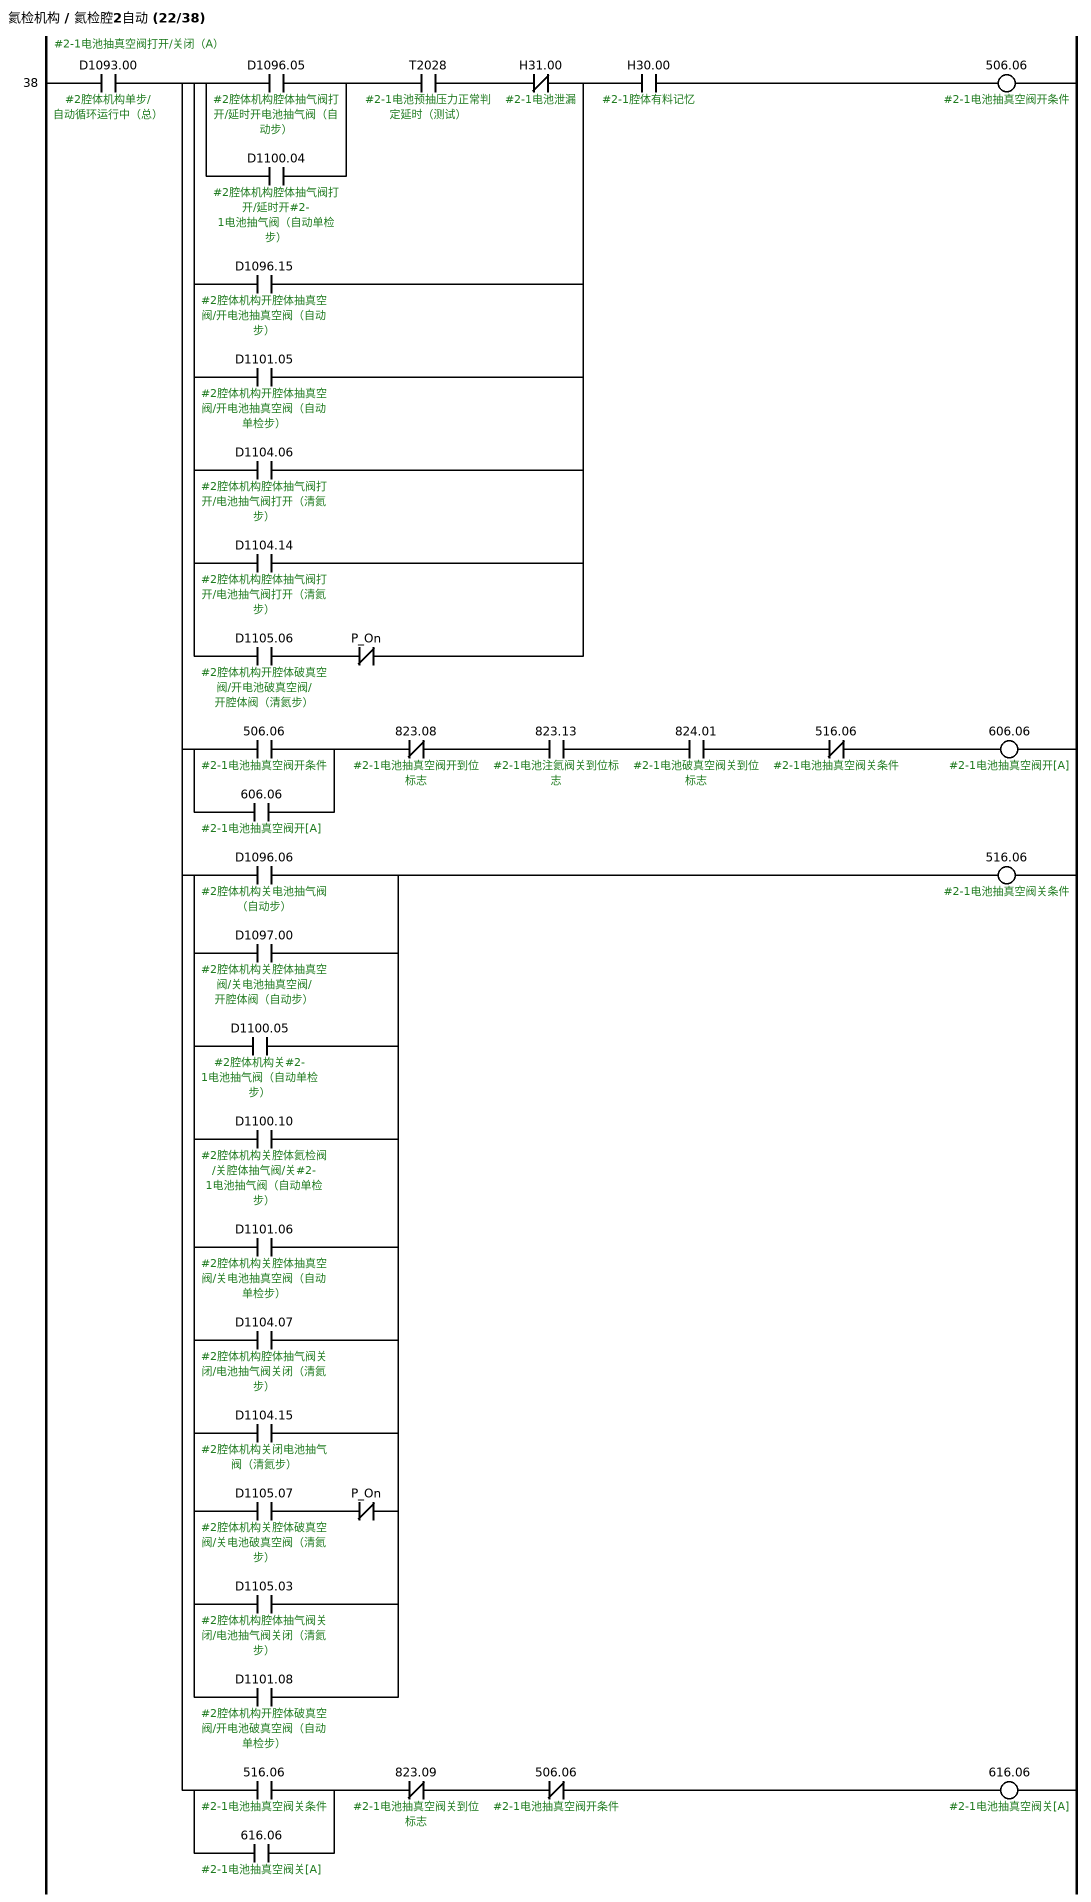
; [picture p264: 氦检机构 / 氦检腔2自动, rungs 38-38]
; rung 38: #2-1电池抽真空阀打开/关闭（A）
LD D1093.00  ; #2腔体机构单步/自动循环运行中（总）
OUT TR0
LD D1096.05  ; #2腔体机构腔体抽气阀打开/延时开电池抽气阀（自动步）
OR D1100.04  ; #2腔体机构腔体抽气阀打开/延时开#2-1电池抽气阀（自动单检步）
AND T2028  ; #2-1电池预抽压力正常判定延时（测试）
ANDNOT H31.00  ; #2-1电池泄漏
OR D1096.15  ; #2腔体机构开腔体抽真空阀/开电池抽真空阀（自动步）
OR D1101.05  ; #2腔体机构开腔体抽真空阀/开电池抽真空阀（自动单检步）
OR D1104.06  ; #2腔体机构腔体抽气阀打开/电池抽气阀打开（清氦步）
OR D1104.14  ; #2腔体机构腔体抽气阀打开/电池抽气阀打开（清氦步）
LD D1105.06  ; #2腔体机构开腔体破真空阀/开电池破真空阀/开腔体阀（清氦步）
ANDNOT P_On
ORLD
ANDLD
AND H30.00  ; #2-1腔体有料记忆
OUT 506.06  ; #2-1电池抽真空阀开条件
LD TR0
LD 506.06  ; #2-1电池抽真空阀开条件
OR 606.06  ; #2-1电池抽真空阀开[A]
ANDLD
ANDNOT 823.08  ; #2-1电池抽真空阀开到位标志
AND 823.13  ; #2-1电池注氦阀关到位标志
AND 824.01  ; #2-1电池破真空阀关到位标志
ANDNOT 516.06  ; #2-1电池抽真空阀关条件
OUT 606.06  ; #2-1电池抽真空阀开[A]
LD TR0
LD D1096.06  ; #2腔体机构关电池抽气阀（自动步）
OR D1097.00  ; #2腔体机构关腔体抽真空阀/关电池抽真空阀/开腔体阀（自动步）
OR D1100.05  ; #2腔体机构关#2-1电池抽气阀（自动单检步）
OR D1100.10  ; #2腔体机构关腔体氦检阀/关腔体抽气阀/关#2-1电池抽气阀（自动单检步）
OR D1101.06  ; #2腔体机构关腔体抽真空阀/关电池抽真空阀（自动单检步）
OR D1104.07  ; #2腔体机构腔体抽气阀关闭/电池抽气阀关闭（清氦步）
OR D1104.15  ; #2腔体机构关闭电池抽气阀（清氦步）
LD D1105.07  ; #2腔体机构关腔体破真空阀/关电池破真空阀（清氦步）
ANDNOT P_On
ORLD
OR D1105.03  ; #2腔体机构腔体抽气阀关闭/电池抽气阀关闭（清氦步）
OR D1101.08  ; #2腔体机构开腔体破真空阀/开电池破真空阀（自动单检步）
ANDLD
OUT 516.06  ; #2-1电池抽真空阀关条件
LD TR0
LD 516.06  ; #2-1电池抽真空阀关条件
OR 616.06  ; #2-1电池抽真空阀关[A]
ANDLD
ANDNOT 823.09  ; #2-1电池抽真空阀关到位标志
ANDNOT 506.06  ; #2-1电池抽真空阀开条件
OUT 616.06  ; #2-1电池抽真空阀关[A]

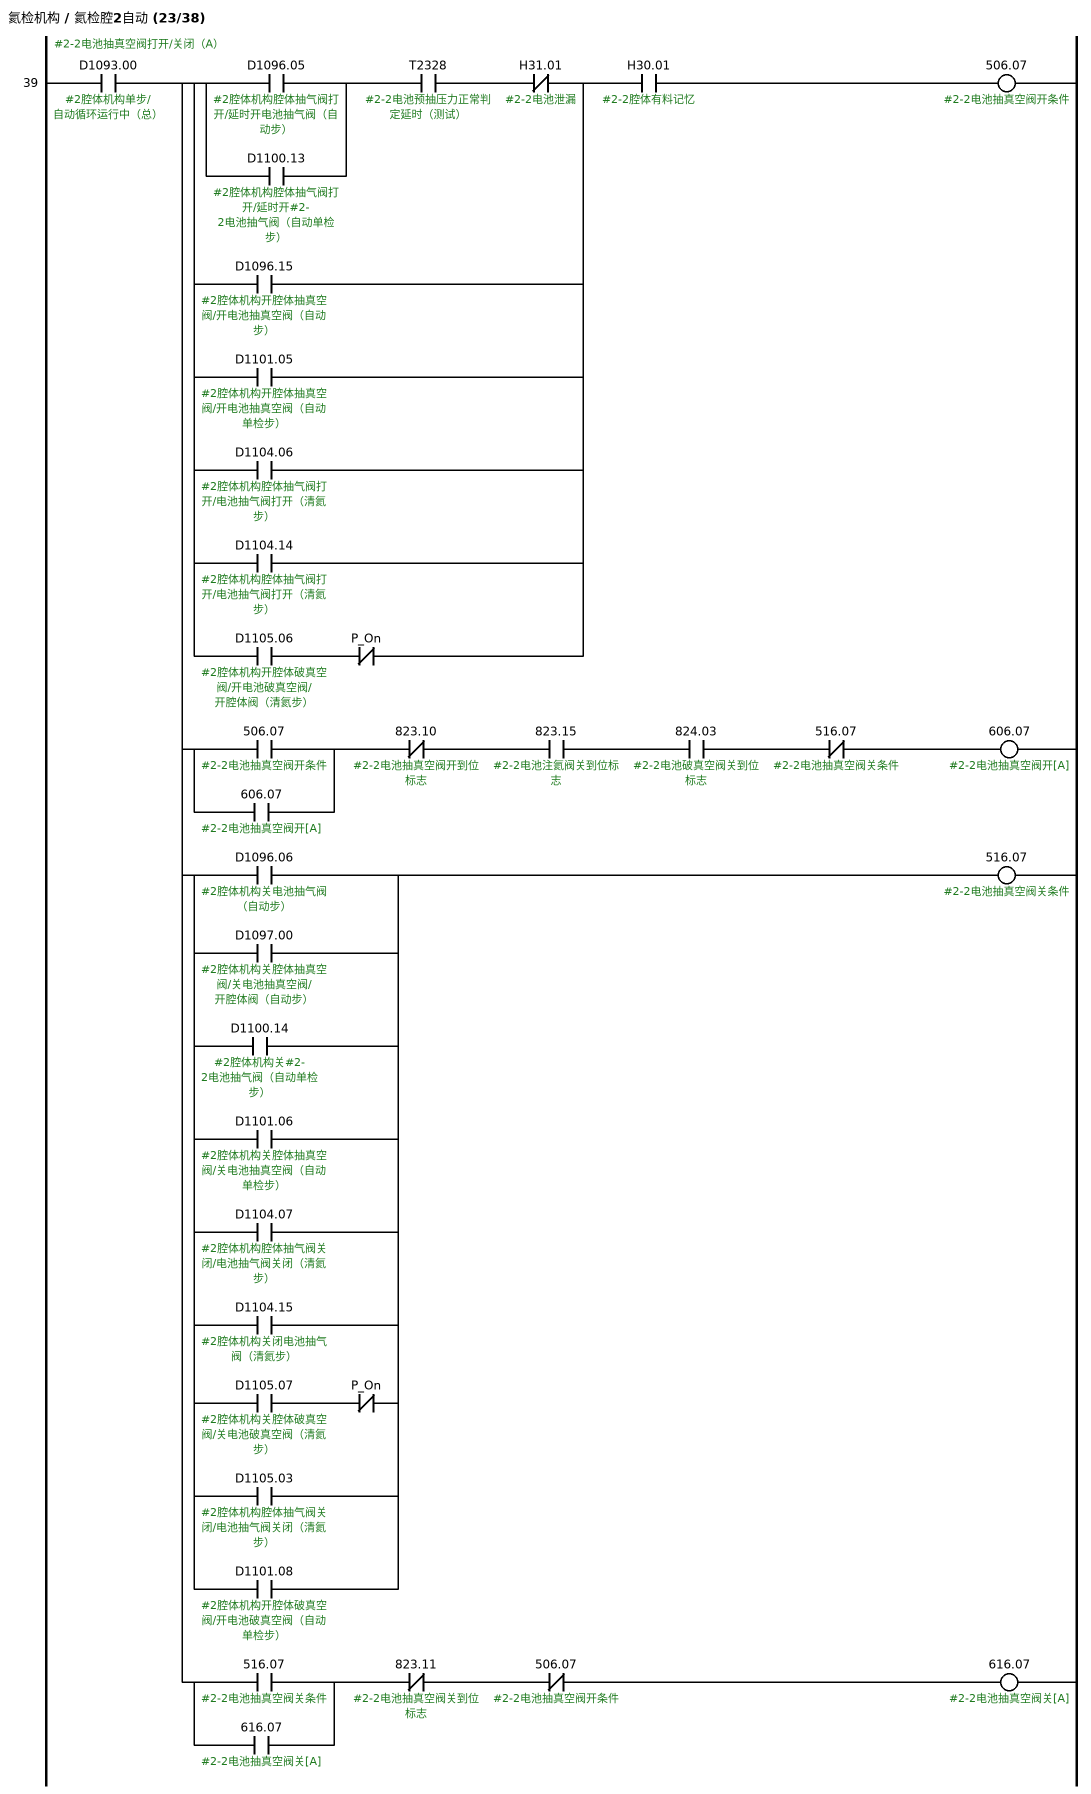
; rung 39: #2-2电池抽真空阀打开/关闭（A）
LD D1093.00  ; #2腔体机构单步/自动循环运行中（总）
OUT TR0
LD D1096.05  ; #2腔体机构腔体抽气阀打开/延时开电池抽气阀（自动步）
OR D1100.13  ; #2腔体机构腔体抽气阀打开/延时开#2-2电池抽气阀（自动单检步）
AND T2328  ; #2-2电池预抽压力正常判定延时（测试）
ANDNOT H31.01  ; #2-2电池泄漏
OR D1096.15  ; #2腔体机构开腔体抽真空阀/开电池抽真空阀（自动步）
OR D1101.05  ; #2腔体机构开腔体抽真空阀/开电池抽真空阀（自动单检步）
OR D1104.06  ; #2腔体机构腔体抽气阀打开/电池抽气阀打开（清氦步）
OR D1104.14  ; #2腔体机构腔体抽气阀打开/电池抽气阀打开（清氦步）
LD D1105.06  ; #2腔体机构开腔体破真空阀/开电池破真空阀/开腔体阀（清氦步）
ANDNOT P_On
ORLD
ANDLD
AND H30.01  ; #2-2腔体有料记忆
OUT 506.07  ; #2-2电池抽真空阀开条件
LD TR0
LD 506.07  ; #2-2电池抽真空阀开条件
OR 606.07  ; #2-2电池抽真空阀开[A]
ANDLD
ANDNOT 823.10  ; #2-2电池抽真空阀开到位标志
AND 823.15  ; #2-2电池注氦阀关到位标志
AND 824.03  ; #2-2电池破真空阀关到位标志
ANDNOT 516.07  ; #2-2电池抽真空阀关条件
OUT 606.07  ; #2-2电池抽真空阀开[A]
LD TR0
LD D1096.06  ; #2腔体机构关电池抽气阀（自动步）
OR D1097.00  ; #2腔体机构关腔体抽真空阀/关电池抽真空阀/开腔体阀（自动步）
OR D1100.14  ; #2腔体机构关#2-2电池抽气阀（自动单检步）
OR D1101.06  ; #2腔体机构关腔体抽真空阀/关电池抽真空阀（自动单检步）
OR D1104.07  ; #2腔体机构腔体抽气阀关闭/电池抽气阀关闭（清氦步）
OR D1104.15  ; #2腔体机构关闭电池抽气阀（清氦步）
LD D1105.07  ; #2腔体机构关腔体破真空阀/关电池破真空阀（清氦步）
ANDNOT P_On
ORLD
OR D1105.03  ; #2腔体机构腔体抽气阀关闭/电池抽气阀关闭（清氦步）
OR D1101.08  ; #2腔体机构开腔体破真空阀/开电池破真空阀（自动单检步）
ANDLD
OUT 516.07  ; #2-2电池抽真空阀关条件
LD TR0
LD 516.07  ; #2-2电池抽真空阀关条件
OR 616.07  ; #2-2电池抽真空阀关[A]
ANDLD
ANDNOT 823.11  ; #2-2电池抽真空阀关到位标志
ANDNOT 506.07  ; #2-2电池抽真空阀开条件
OUT 616.07  ; #2-2电池抽真空阀关[A]

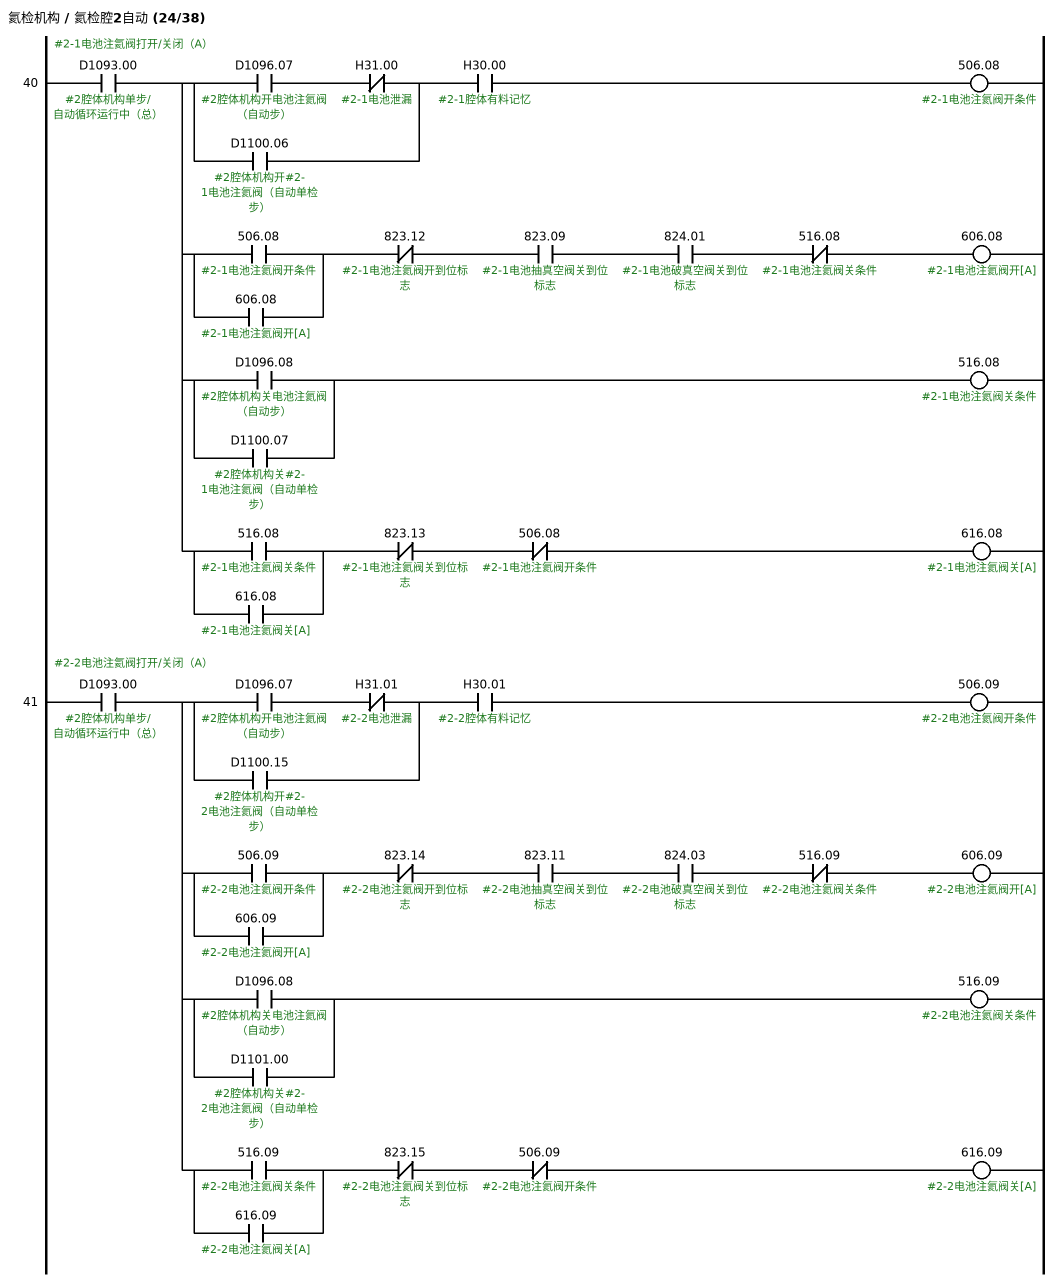
; rung 40: #2-1电池注氦阀打开/关闭（A）
LD D1093.00  ; #2腔体机构单步/自动循环运行中（总）
OUT TR0
LD D1096.07  ; #2腔体机构开电池注氦阀（自动步）
ANDNOT H31.00  ; #2-1电池泄漏
OR D1100.06  ; #2腔体机构开#2-1电池注氦阀（自动单检步）
ANDLD
AND H30.00  ; #2-1腔体有料记忆
OUT 506.08  ; #2-1电池注氦阀开条件
LD TR0
LD 506.08  ; #2-1电池注氦阀开条件
OR 606.08  ; #2-1电池注氦阀开[A]
ANDLD
ANDNOT 823.12  ; #2-1电池注氦阀开到位标志
AND 823.09  ; #2-1电池抽真空阀关到位标志
AND 824.01  ; #2-1电池破真空阀关到位标志
ANDNOT 516.08  ; #2-1电池注氦阀关条件
OUT 606.08  ; #2-1电池注氦阀开[A]
LD TR0
LD D1096.08  ; #2腔体机构关电池注氦阀（自动步）
OR D1100.07  ; #2腔体机构关#2-1电池注氦阀（自动单检步）
ANDLD
OUT 516.08  ; #2-1电池注氦阀关条件
LD TR0
LD 516.08  ; #2-1电池注氦阀关条件
OR 616.08  ; #2-1电池注氦阀关[A]
ANDLD
ANDNOT 823.13  ; #2-1电池注氦阀关到位标志
ANDNOT 506.08  ; #2-1电池注氦阀开条件
OUT 616.08  ; #2-1电池注氦阀关[A]
; rung 41: #2-2电池注氦阀打开/关闭（A）
LD D1093.00  ; #2腔体机构单步/自动循环运行中（总）
OUT TR0
LD D1096.07  ; #2腔体机构开电池注氦阀（自动步）
ANDNOT H31.01  ; #2-2电池泄漏
OR D1100.15  ; #2腔体机构开#2-2电池注氦阀（自动单检步）
ANDLD
AND H30.01  ; #2-2腔体有料记忆
OUT 506.09  ; #2-2电池注氦阀开条件
LD TR0
LD 506.09  ; #2-2电池注氦阀开条件
OR 606.09  ; #2-2电池注氦阀开[A]
ANDLD
ANDNOT 823.14  ; #2-2电池注氦阀开到位标志
AND 823.11  ; #2-2电池抽真空阀关到位标志
AND 824.03  ; #2-2电池破真空阀关到位标志
ANDNOT 516.09  ; #2-2电池注氦阀关条件
OUT 606.09  ; #2-2电池注氦阀开[A]
LD TR0
LD D1096.08  ; #2腔体机构关电池注氦阀（自动步）
OR D1101.00  ; #2腔体机构关#2-2电池注氦阀（自动单检步）
ANDLD
OUT 516.09  ; #2-2电池注氦阀关条件
LD TR0
LD 516.09  ; #2-2电池注氦阀关条件
OR 616.09  ; #2-2电池注氦阀关[A]
ANDLD
ANDNOT 823.15  ; #2-2电池注氦阀关到位标志
ANDNOT 506.09  ; #2-2电池注氦阀开条件
OUT 616.09  ; #2-2电池注氦阀关[A]

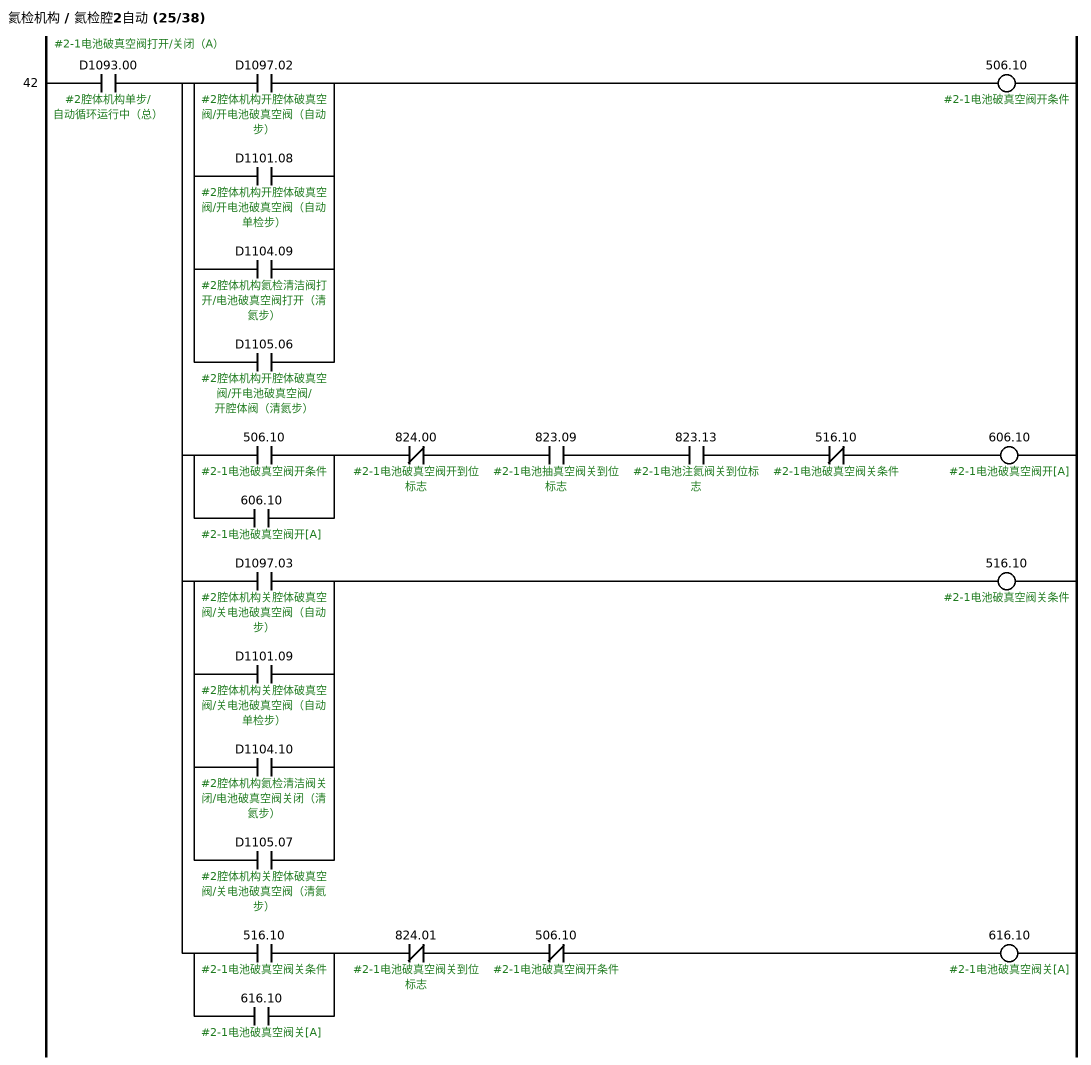
; rung 42: #2-1电池破真空阀打开/关闭（A）
LD D1093.00  ; #2腔体机构单步/自动循环运行中（总）
OUT TR0
LD D1097.02  ; #2腔体机构开腔体破真空阀/开电池破真空阀（自动步）
OR D1101.08  ; #2腔体机构开腔体破真空阀/开电池破真空阀（自动单检步）
OR D1104.09  ; #2腔体机构氦检清洁阀打开/电池破真空阀打开（清氦步）
OR D1105.06  ; #2腔体机构开腔体破真空阀/开电池破真空阀/开腔体阀（清氦步）
ANDLD
OUT 506.10  ; #2-1电池破真空阀开条件
LD TR0
LD 506.10  ; #2-1电池破真空阀开条件
OR 606.10  ; #2-1电池破真空阀开[A]
ANDLD
ANDNOT 824.00  ; #2-1电池破真空阀开到位标志
AND 823.09  ; #2-1电池抽真空阀关到位标志
AND 823.13  ; #2-1电池注氦阀关到位标志
ANDNOT 516.10  ; #2-1电池破真空阀关条件
OUT 606.10  ; #2-1电池破真空阀开[A]
LD TR0
LD D1097.03  ; #2腔体机构关腔体破真空阀/关电池破真空阀（自动步）
OR D1101.09  ; #2腔体机构关腔体破真空阀/关电池破真空阀（自动单检步）
OR D1104.10  ; #2腔体机构氦检清洁阀关闭/电池破真空阀关闭（清氦步）
OR D1105.07  ; #2腔体机构关腔体破真空阀/关电池破真空阀（清氦步）
ANDLD
OUT 516.10  ; #2-1电池破真空阀关条件
LD TR0
LD 516.10  ; #2-1电池破真空阀关条件
OR 616.10  ; #2-1电池破真空阀关[A]
ANDLD
ANDNOT 824.01  ; #2-1电池破真空阀关到位标志
ANDNOT 506.10  ; #2-1电池破真空阀开条件
OUT 616.10  ; #2-1电池破真空阀关[A]

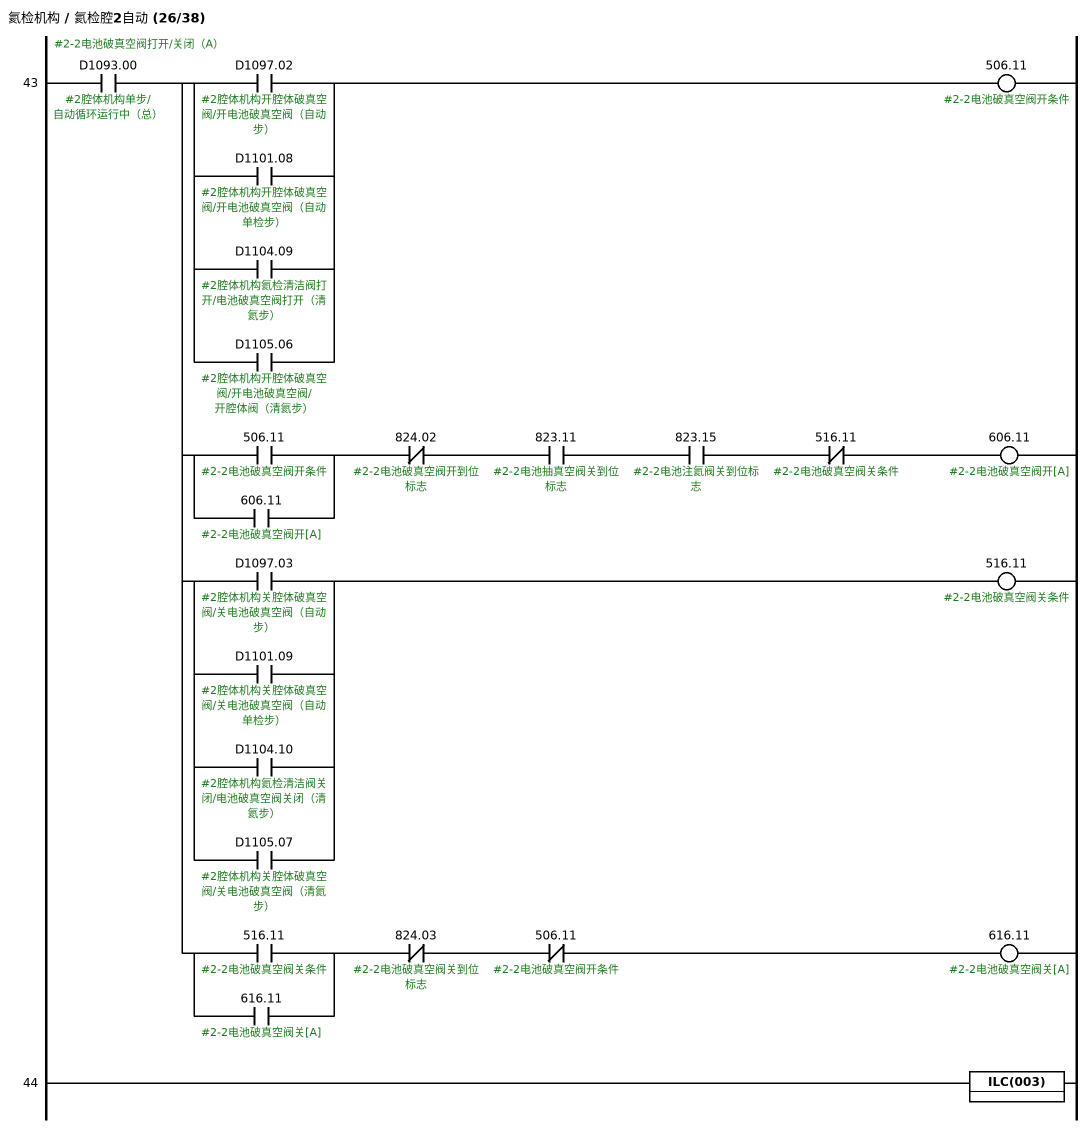
; rung 43: #2-2电池破真空阀打开/关闭（A）
LD D1093.00  ; #2腔体机构单步/自动循环运行中（总）
OUT TR0
LD D1097.02  ; #2腔体机构开腔体破真空阀/开电池破真空阀（自动步）
OR D1101.08  ; #2腔体机构开腔体破真空阀/开电池破真空阀（自动单检步）
OR D1104.09  ; #2腔体机构氦检清洁阀打开/电池破真空阀打开（清氦步）
OR D1105.06  ; #2腔体机构开腔体破真空阀/开电池破真空阀/开腔体阀（清氦步）
ANDLD
OUT 506.11  ; #2-2电池破真空阀开条件
LD TR0
LD 506.11  ; #2-2电池破真空阀开条件
OR 606.11  ; #2-2电池破真空阀开[A]
ANDLD
ANDNOT 824.02  ; #2-2电池破真空阀开到位标志
AND 823.11  ; #2-2电池抽真空阀关到位标志
AND 823.15  ; #2-2电池注氦阀关到位标志
ANDNOT 516.11  ; #2-2电池破真空阀关条件
OUT 606.11  ; #2-2电池破真空阀开[A]
LD TR0
LD D1097.03  ; #2腔体机构关腔体破真空阀/关电池破真空阀（自动步）
OR D1101.09  ; #2腔体机构关腔体破真空阀/关电池破真空阀（自动单检步）
OR D1104.10  ; #2腔体机构氦检清洁阀关闭/电池破真空阀关闭（清氦步）
OR D1105.07  ; #2腔体机构关腔体破真空阀/关电池破真空阀（清氦步）
ANDLD
OUT 516.11  ; #2-2电池破真空阀关条件
LD TR0
LD 516.11  ; #2-2电池破真空阀关条件
OR 616.11  ; #2-2电池破真空阀关[A]
ANDLD
ANDNOT 824.03  ; #2-2电池破真空阀关到位标志
ANDNOT 506.11  ; #2-2电池破真空阀开条件
OUT 616.11  ; #2-2电池破真空阀关[A]
; rung 44
ILC(003)

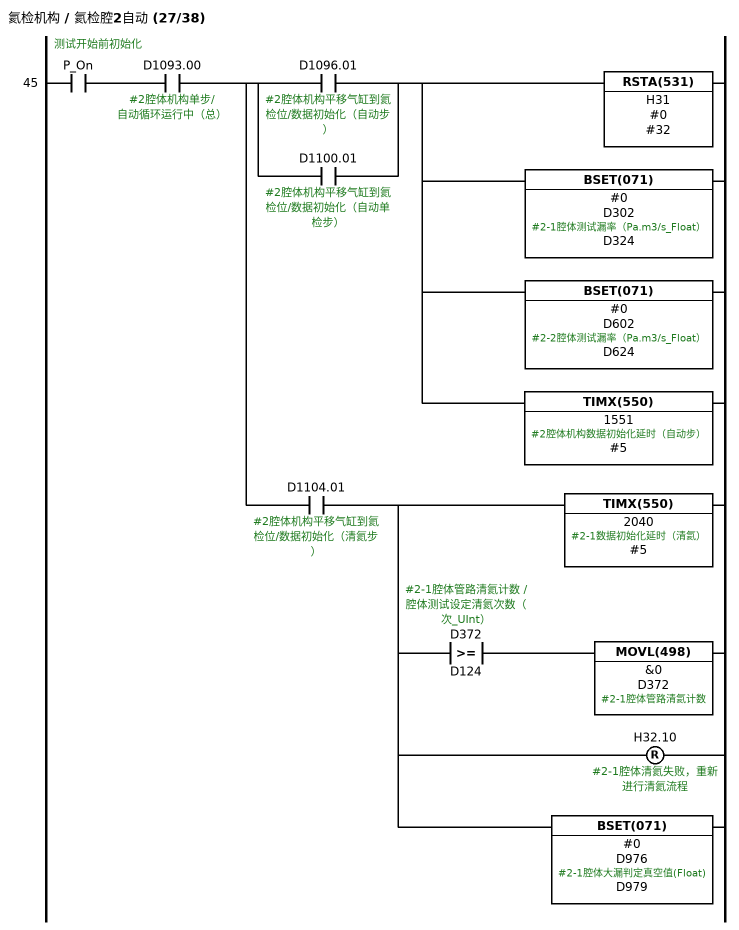
; rung 45: 测试开始前初始化
LD P_On
AND D1093.00  ; #2腔体机构单步/自动循环运行中（总）
OUT TR0
LD D1096.01  ; #2腔体机构平移气缸到氦检位/数据初始化（自动步）
OR D1100.01  ; #2腔体机构平移气缸到氦检位/数据初始化（自动单检步）
ANDLD
RSTA(531) H31 #0 #32
BSET(071) #0 D302 D324  ; #2-1腔体测试漏率（Pa.m3/s_Float）
BSET(071) #0 D602 D624  ; #2-2腔体测试漏率（Pa.m3/s_Float）
TIMX(550) 1551 #5  ; #2腔体机构数据初始化延时（自动步）
LD TR0
AND D1104.01  ; #2腔体机构平移气缸到氦检位/数据初始化（清氦步）
OUT TR0
TIMX(550) 2040 #5  ; #2-1数据初始化延时（清氦）
AND>=(325) D372 D124  ; #2-1腔体管路清氦计数, 腔体测试设定清氦次数（次_UInt）
MOVL(498) &0 D372  ; #2-1腔体管路清氦计数
LD TR0
RSET H32.10  ; #2-1腔体清氦失败，重新进行清氦流程
BSET(071) #0 D976 D979  ; #2-1腔体大漏判定真空值(Float)

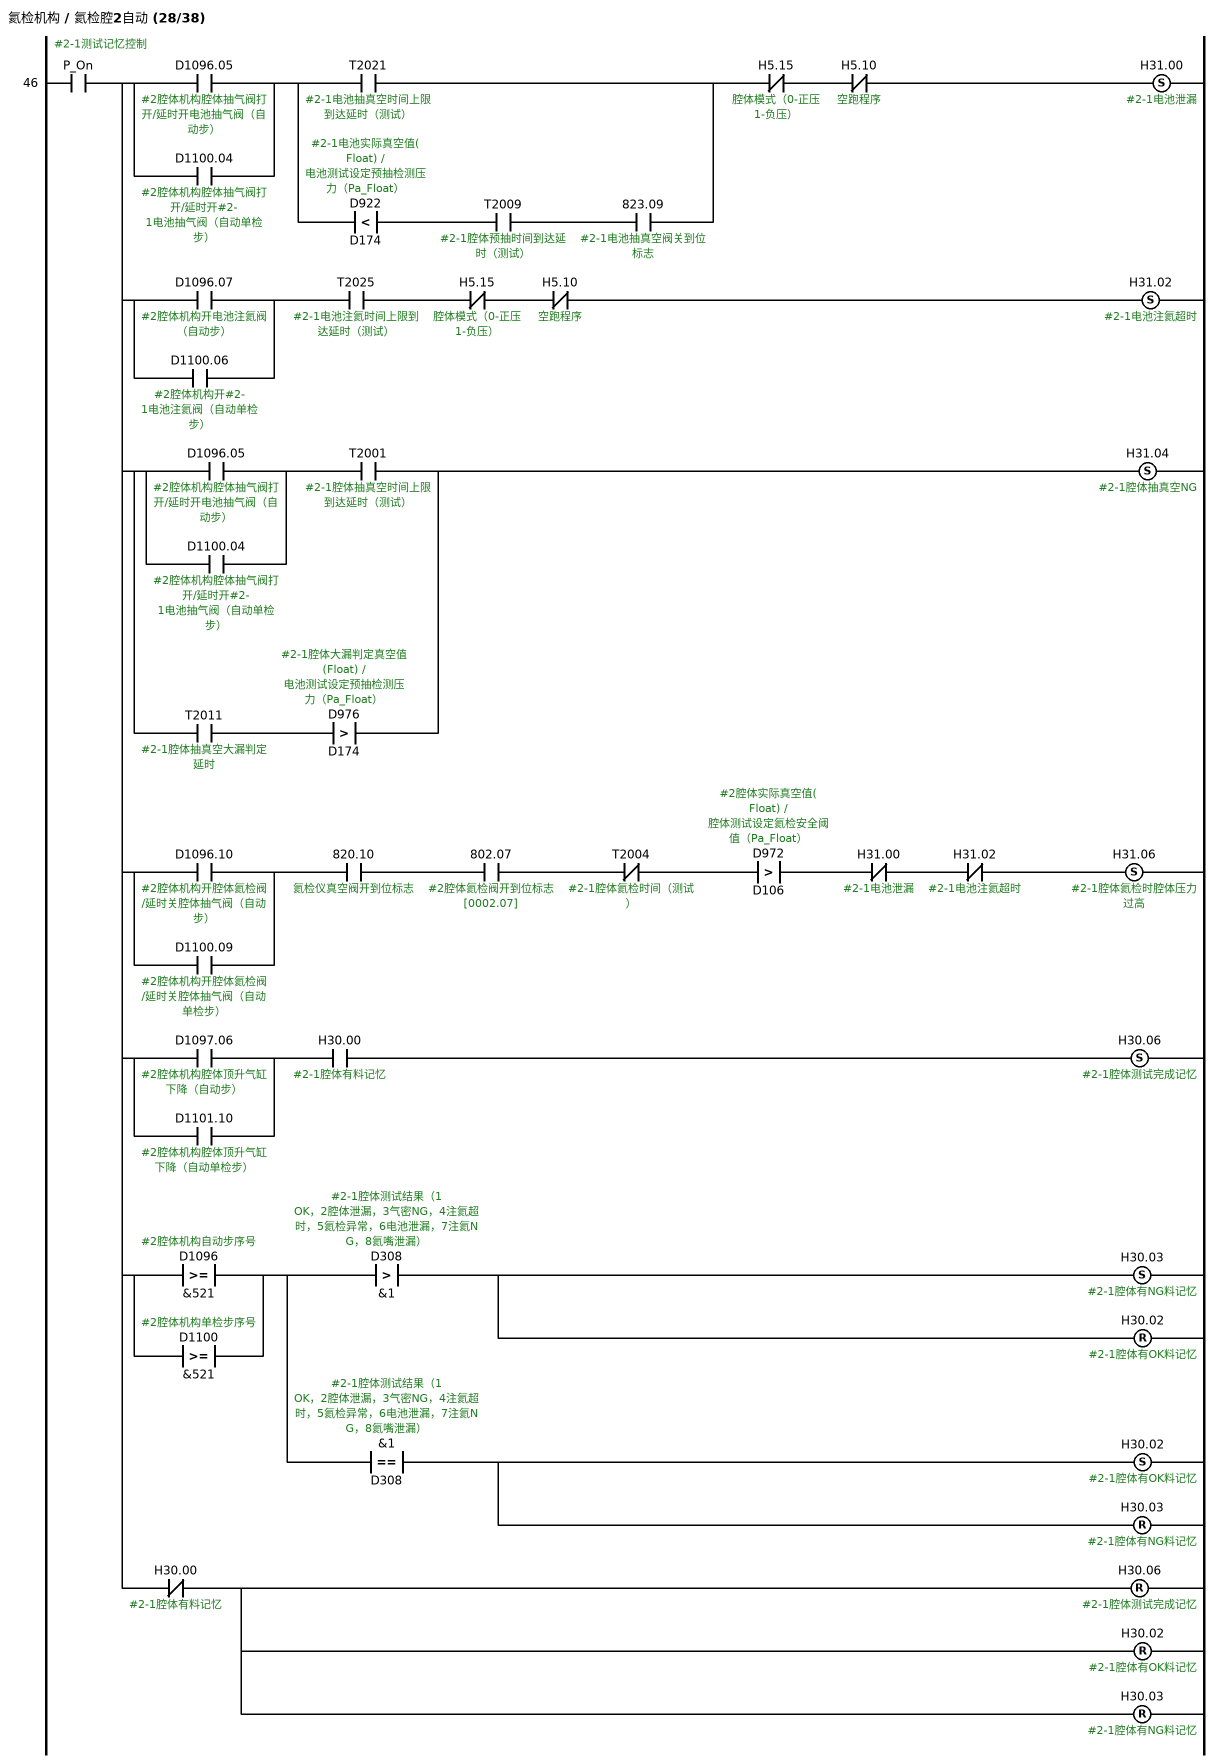
; rung 46: #2-1测试记忆控制
LD P_On
OUT TR0
LD D1096.05  ; #2腔体机构腔体抽气阀打开/延时开电池抽气阀（自动步）
OR D1100.04  ; #2腔体机构腔体抽气阀打开/延时开#2-1电池抽气阀（自动单检步）
ANDLD
LD T2021  ; #2-1电池抽真空时间上限到达延时（测试）
LD<F(331) D922 D174  ; #2-1电池实际真空值(Float), 电池测试设定预抽检测压力（Pa_Float）
AND T2009  ; #2-1腔体预抽时间到达延时（测试）
AND 823.09  ; #2-1电池抽真空阀关到位标志
ORLD
ANDLD
ANDNOT H5.15  ; 腔体模式（0-正压 1-负压）
ANDNOT H5.10  ; 空跑程序
SET H31.00  ; #2-1电池泄漏
LD TR0
LD D1096.07  ; #2腔体机构开电池注氦阀（自动步）
OR D1100.06  ; #2腔体机构开#2-1电池注氦阀（自动单检步）
ANDLD
AND T2025  ; #2-1电池注氦时间上限到达延时（测试）
ANDNOT H5.15  ; 腔体模式（0-正压 1-负压）
ANDNOT H5.10  ; 空跑程序
SET H31.02  ; #2-1电池注氦超时
LD TR0
LD D1096.05  ; #2腔体机构腔体抽气阀打开/延时开电池抽气阀（自动步）
OR D1100.04  ; #2腔体机构腔体抽气阀打开/延时开#2-1电池抽气阀（自动单检步）
AND T2001  ; #2-1腔体抽真空时间上限到达延时（测试）
LD T2011  ; #2-1腔体抽真空大漏判定延时
AND>F(333) D976 D174  ; #2-1腔体大漏判定真空值(Float), 电池测试设定预抽检测压力（Pa_Float）
ORLD
ANDLD
SET H31.04  ; #2-1腔体抽真空NG
LD TR0
LD D1096.10  ; #2腔体机构开腔体氦检阀/延时关腔体抽气阀（自动步）
OR D1100.09  ; #2腔体机构开腔体氦检阀/延时关腔体抽气阀（自动单检步）
ANDLD
AND 820.10  ; 氦检仪真空阀开到位标志
AND 802.07  ; #2腔体氦检阀开到位标志[0002.07]
ANDNOT T2004  ; #2-1腔体氦检时间（测试）
AND>F(333) D972 D106  ; #2腔体实际真空值(Float), 腔体测试设定氦检安全阈值（Pa_Float）
ANDNOT H31.00  ; #2-1电池泄漏
ANDNOT H31.02  ; #2-1电池注氦超时
SET H31.06  ; #2-1腔体氦检时腔体压力过高
LD TR0
LD D1097.06  ; #2腔体机构腔体顶升气缸下降（自动步）
OR D1101.10  ; #2腔体机构腔体顶升气缸下降（自动单检步）
ANDLD
AND H30.00  ; #2-1腔体有料记忆
SET H30.06  ; #2-1腔体测试完成记忆
LD TR0
LD>=L(326) D1096 &521  ; #2腔体机构自动步序号
OR>=L(326) D1100 &521  ; #2腔体机构单检步序号
ANDLD
OUT TR1
AND>(320) D308 &1  ; #2-1腔体测试结果（1 OK，2腔体泄漏，3气密NG，4注氦超时，5氦检异常，6电池泄漏，7注氦NG，8氦嘴泄漏）
SET H30.03  ; #2-1腔体有NG料记忆
RSET H30.02  ; #2-1腔体有OK料记忆
LD TR1
AND=(300) &1 D308  ; #2-1腔体测试结果（1 OK，2腔体泄漏，3气密NG，4注氦超时，5氦检异常，6电池泄漏，7注氦NG，8氦嘴泄漏）
SET H30.02  ; #2-1腔体有OK料记忆
RSET H30.03  ; #2-1腔体有NG料记忆
LD TR0
ANDNOT H30.00  ; #2-1腔体有料记忆
RSET H30.06  ; #2-1腔体测试完成记忆
RSET H30.02  ; #2-1腔体有OK料记忆
RSET H30.03  ; #2-1腔体有NG料记忆

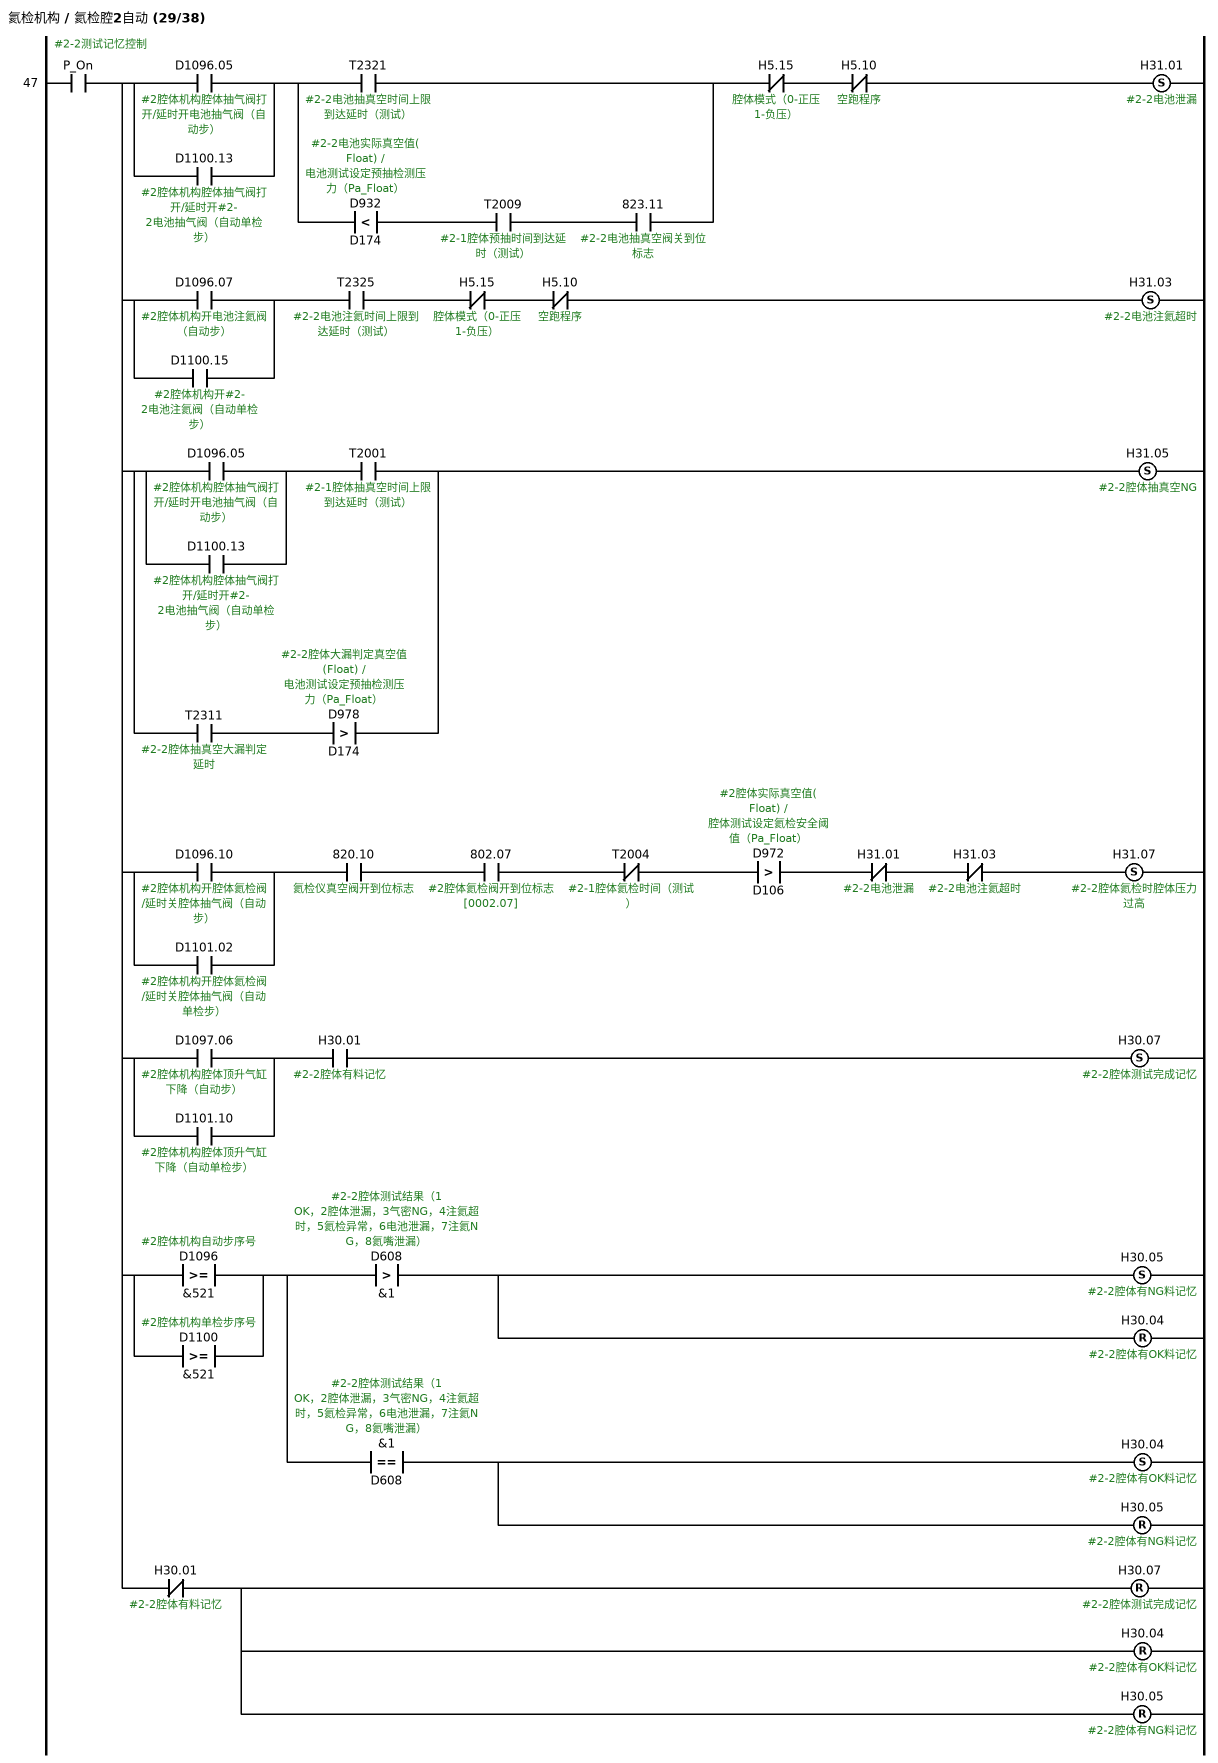
; rung 47: #2-2测试记忆控制
LD P_On
OUT TR0
LD D1096.05  ; #2腔体机构腔体抽气阀打开/延时开电池抽气阀（自动步）
OR D1100.13  ; #2腔体机构腔体抽气阀打开/延时开#2-2电池抽气阀（自动单检步）
ANDLD
LD T2321  ; #2-2电池抽真空时间上限到达延时（测试）
LD<F(331) D932 D174  ; #2-2电池实际真空值(Float), 电池测试设定预抽检测压力（Pa_Float）
AND T2009  ; #2-1腔体预抽时间到达延时（测试）
AND 823.11  ; #2-2电池抽真空阀关到位标志
ORLD
ANDLD
ANDNOT H5.15  ; 腔体模式（0-正压 1-负压）
ANDNOT H5.10  ; 空跑程序
SET H31.01  ; #2-2电池泄漏
LD TR0
LD D1096.07  ; #2腔体机构开电池注氦阀（自动步）
OR D1100.15  ; #2腔体机构开#2-2电池注氦阀（自动单检步）
ANDLD
AND T2325  ; #2-2电池注氦时间上限到达延时（测试）
ANDNOT H5.15  ; 腔体模式（0-正压 1-负压）
ANDNOT H5.10  ; 空跑程序
SET H31.03  ; #2-2电池注氦超时
LD TR0
LD D1096.05  ; #2腔体机构腔体抽气阀打开/延时开电池抽气阀（自动步）
OR D1100.13  ; #2腔体机构腔体抽气阀打开/延时开#2-2电池抽气阀（自动单检步）
AND T2001  ; #2-1腔体抽真空时间上限到达延时（测试）
LD T2311  ; #2-2腔体抽真空大漏判定延时
AND>F(333) D978 D174  ; #2-2腔体大漏判定真空值(Float), 电池测试设定预抽检测压力（Pa_Float）
ORLD
ANDLD
SET H31.05  ; #2-2腔体抽真空NG
LD TR0
LD D1096.10  ; #2腔体机构开腔体氦检阀/延时关腔体抽气阀（自动步）
OR D1101.02  ; #2腔体机构开腔体氦检阀/延时关腔体抽气阀（自动单检步）
ANDLD
AND 820.10  ; 氦检仪真空阀开到位标志
AND 802.07  ; #2腔体氦检阀开到位标志[0002.07]
ANDNOT T2004  ; #2-1腔体氦检时间（测试）
AND>F(333) D972 D106  ; #2腔体实际真空值(Float), 腔体测试设定氦检安全阈值（Pa_Float）
ANDNOT H31.01  ; #2-2电池泄漏
ANDNOT H31.03  ; #2-2电池注氦超时
SET H31.07  ; #2-2腔体氦检时腔体压力过高
LD TR0
LD D1097.06  ; #2腔体机构腔体顶升气缸下降（自动步）
OR D1101.10  ; #2腔体机构腔体顶升气缸下降（自动单检步）
ANDLD
AND H30.01  ; #2-2腔体有料记忆
SET H30.07  ; #2-2腔体测试完成记忆
LD TR0
LD>=L(326) D1096 &521  ; #2腔体机构自动步序号
OR>=L(326) D1100 &521  ; #2腔体机构单检步序号
ANDLD
OUT TR1
AND>(320) D608 &1  ; #2-2腔体测试结果（1 OK，2腔体泄漏，3气密NG，4注氦超时，5氦检异常，6电池泄漏，7注氦NG，8氦嘴泄漏）
SET H30.05  ; #2-2腔体有NG料记忆
RSET H30.04  ; #2-2腔体有OK料记忆
LD TR1
AND=(300) &1 D608  ; #2-2腔体测试结果（1 OK，2腔体泄漏，3气密NG，4注氦超时，5氦检异常，6电池泄漏，7注氦NG，8氦嘴泄漏）
SET H30.04  ; #2-2腔体有OK料记忆
RSET H30.05  ; #2-2腔体有NG料记忆
LD TR0
ANDNOT H30.01  ; #2-2腔体有料记忆
RSET H30.07  ; #2-2腔体测试完成记忆
RSET H30.04  ; #2-2腔体有OK料记忆
RSET H30.05  ; #2-2腔体有NG料记忆

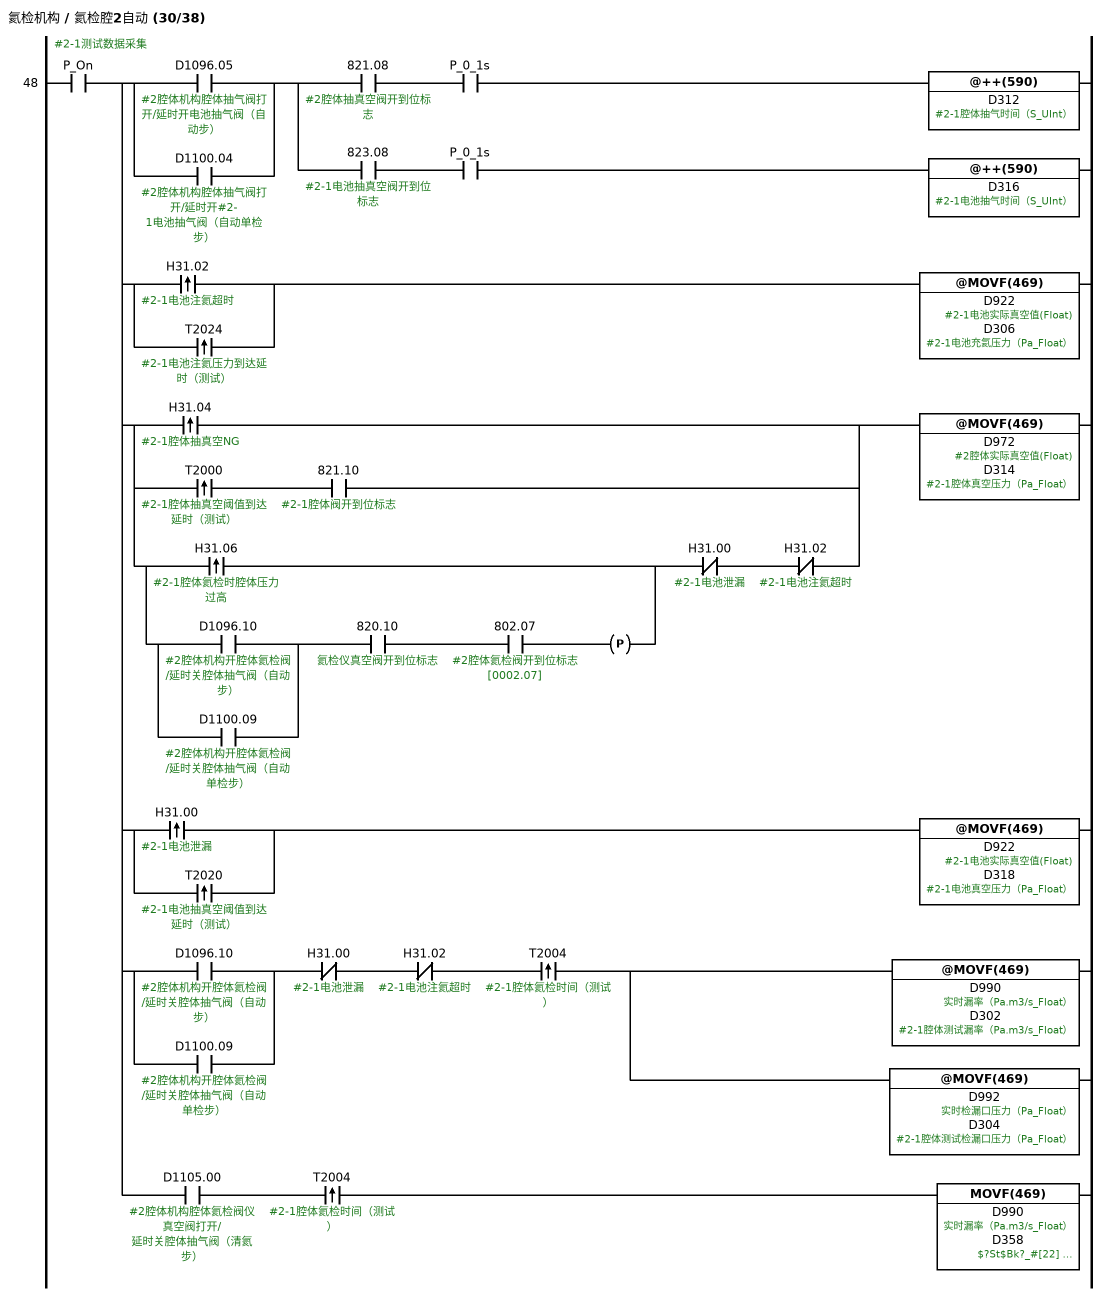
; rung 48: #2-1测试数据采集
LD P_On
OUT TR0
LD D1096.05  ; #2腔体机构腔体抽气阀打开/延时开电池抽气阀（自动步）
OR D1100.04  ; #2腔体机构腔体抽气阀打开/延时开#2-1电池抽气阀（自动单检步）
ANDLD
OUT TR1
AND 821.08  ; #2腔体抽真空阀开到位标志
AND P_0_1s
@++(590) D312  ; #2-1腔体抽气时间（S_UInt）
LD TR1
AND 823.08  ; #2-1电池抽真空阀开到位标志
AND P_0_1s
@++(590) D316  ; #2-1电池抽气时间（S_UInt）
LD TR0
@LD H31.02  ; #2-1电池注氦超时
@OR T2024  ; #2-1电池注氦压力到达延时（测试）
ANDLD
@MOVF(469) D922 D306  ; #2-1电池实际真空值(Float), #2-1电池充氦压力（Pa_Float）
LD TR0
@LD H31.04  ; #2-1腔体抽真空NG
@LD T2000  ; #2-1腔体抽真空阈值到达延时（测试）
AND 821.10  ; #2-1腔体阀开到位标志
ORLD
@LD H31.06  ; #2-1腔体氦检时腔体压力过高
LD D1096.10  ; #2腔体机构开腔体氦检阀/延时关腔体抽气阀（自动步）
OR D1100.09  ; #2腔体机构开腔体氦检阀/延时关腔体抽气阀（自动单检步）
AND 820.10  ; 氦检仪真空阀开到位标志
AND 802.07  ; #2腔体氦检阀开到位标志[0002.07]
UP(521)
ORLD
ANDNOT H31.00  ; #2-1电池泄漏
ANDNOT H31.02  ; #2-1电池注氦超时
ORLD
ANDLD
@MOVF(469) D972 D314  ; #2腔体实际真空值(Float), #2-1腔体真空压力（Pa_Float）
LD TR0
@LD H31.00  ; #2-1电池泄漏
@OR T2020  ; #2-1电池抽真空阈值到达延时（测试）
ANDLD
@MOVF(469) D922 D318  ; #2-1电池实际真空值(Float), #2-1电池真空压力（Pa_Float）
LD TR0
LD D1096.10  ; #2腔体机构开腔体氦检阀/延时关腔体抽气阀（自动步）
OR D1100.09  ; #2腔体机构开腔体氦检阀/延时关腔体抽气阀（自动单检步）
ANDLD
ANDNOT H31.00  ; #2-1电池泄漏
ANDNOT H31.02  ; #2-1电池注氦超时
@AND T2004  ; #2-1腔体氦检时间（测试）
@MOVF(469) D990 D302  ; 实时漏率（Pa.m3/s_Float）, #2-1腔体测试漏率（Pa.m3/s_Float）
@MOVF(469) D992 D304  ; 实时检漏口压力（Pa_Float）, #2-1腔体测试检漏口压力（Pa_Float）
LD TR0
AND D1105.00  ; #2腔体机构腔体氦检阀仪真空阀打开/延时关腔体抽气阀（清氦步）
@AND T2004  ; #2-1腔体氦检时间（测试）
MOVF(469) D990 D358  ; 实时漏率（Pa.m3/s_Float）, $?St$Bk?_#[22] / #2-1清氦泄漏率（清氦） / $?St$Bk?_#[22]

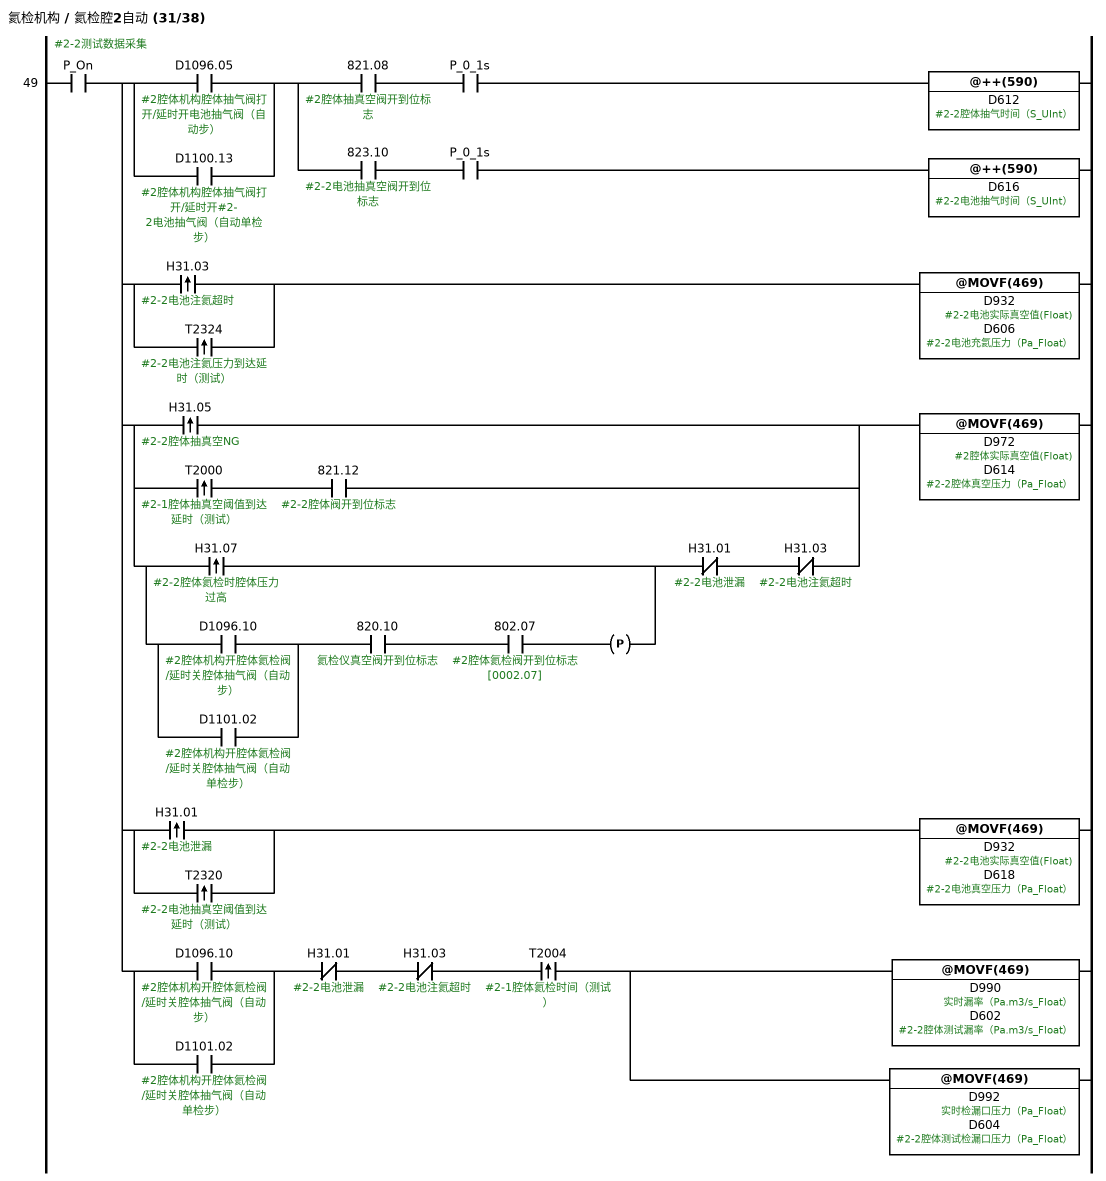
; rung 49: #2-2测试数据采集
LD P_On
OUT TR0
LD D1096.05  ; #2腔体机构腔体抽气阀打开/延时开电池抽气阀（自动步）
OR D1100.13  ; #2腔体机构腔体抽气阀打开/延时开#2-2电池抽气阀（自动单检步）
ANDLD
OUT TR1
AND 821.08  ; #2腔体抽真空阀开到位标志
AND P_0_1s
@++(590) D612  ; #2-2腔体抽气时间（S_UInt）
LD TR1
AND 823.10  ; #2-2电池抽真空阀开到位标志
AND P_0_1s
@++(590) D616  ; #2-2电池抽气时间（S_UInt）
LD TR0
@LD H31.03  ; #2-2电池注氦超时
@OR T2324  ; #2-2电池注氦压力到达延时（测试）
ANDLD
@MOVF(469) D932 D606  ; #2-2电池实际真空值(Float), #2-2电池充氦压力（Pa_Float）
LD TR0
@LD H31.05  ; #2-2腔体抽真空NG
@LD T2000  ; #2-1腔体抽真空阈值到达延时（测试）
AND 821.12  ; #2-2腔体阀开到位标志
ORLD
@LD H31.07  ; #2-2腔体氦检时腔体压力过高
LD D1096.10  ; #2腔体机构开腔体氦检阀/延时关腔体抽气阀（自动步）
OR D1101.02  ; #2腔体机构开腔体氦检阀/延时关腔体抽气阀（自动单检步）
AND 820.10  ; 氦检仪真空阀开到位标志
AND 802.07  ; #2腔体氦检阀开到位标志[0002.07]
UP(521)
ORLD
ANDNOT H31.01  ; #2-2电池泄漏
ANDNOT H31.03  ; #2-2电池注氦超时
ORLD
ANDLD
@MOVF(469) D972 D614  ; #2腔体实际真空值(Float), #2-2腔体真空压力（Pa_Float）
LD TR0
@LD H31.01  ; #2-2电池泄漏
@OR T2320  ; #2-2电池抽真空阈值到达延时（测试）
ANDLD
@MOVF(469) D932 D618  ; #2-2电池实际真空值(Float), #2-2电池真空压力（Pa_Float）
LD TR0
LD D1096.10  ; #2腔体机构开腔体氦检阀/延时关腔体抽气阀（自动步）
OR D1101.02  ; #2腔体机构开腔体氦检阀/延时关腔体抽气阀（自动单检步）
ANDLD
ANDNOT H31.01  ; #2-2电池泄漏
ANDNOT H31.03  ; #2-2电池注氦超时
@AND T2004  ; #2-1腔体氦检时间（测试）
@MOVF(469) D990 D602  ; 实时漏率（Pa.m3/s_Float）, #2-2腔体测试漏率（Pa.m3/s_Float）
@MOVF(469) D992 D604  ; 实时检漏口压力（Pa_Float）, #2-2腔体测试检漏口压力（Pa_Float）

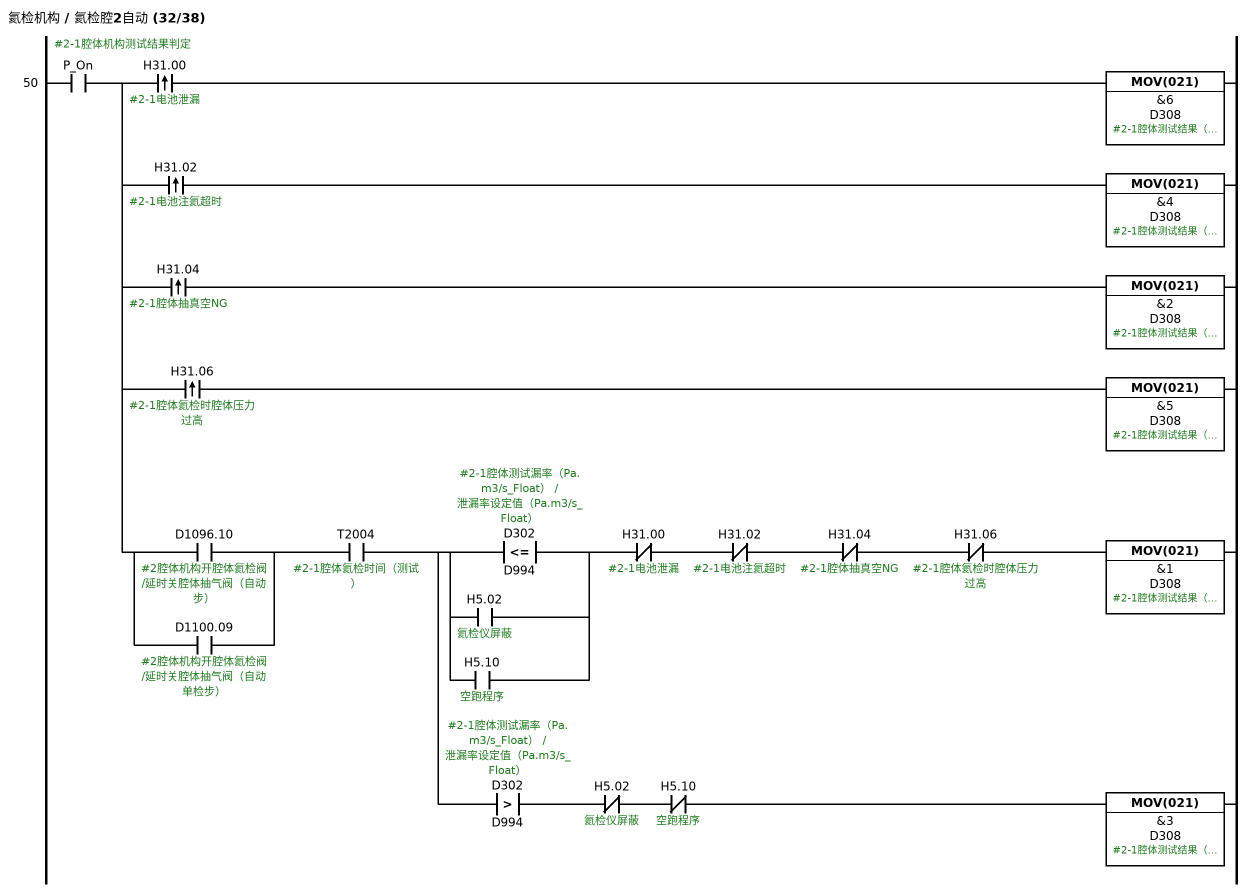
; rung 50: #2-1腔体机构测试结果判定
LD P_On
OUT TR0
@AND H31.00  ; #2-1电池泄漏
MOV(021) &6 D308  ; #2-1腔体测试结果（1 OK，2腔体泄漏，3气密NG，4注氦超时，5氦检异常，6电池泄漏，7注氦NG，8氦嘴泄漏）
LD TR0
@AND H31.02  ; #2-1电池注氦超时
MOV(021) &4 D308  ; #2-1腔体测试结果（1 OK，2腔体泄漏，3气密NG，4注氦超时，5氦检异常，6电池泄漏，7注氦NG，8氦嘴泄漏）
LD TR0
@AND H31.04  ; #2-1腔体抽真空NG
MOV(021) &2 D308  ; #2-1腔体测试结果（1 OK，2腔体泄漏，3气密NG，4注氦超时，5氦检异常，6电池泄漏，7注氦NG，8氦嘴泄漏）
LD TR0
@AND H31.06  ; #2-1腔体氦检时腔体压力过高
MOV(021) &5 D308  ; #2-1腔体测试结果（1 OK，2腔体泄漏，3气密NG，4注氦超时，5氦检异常，6电池泄漏，7注氦NG，8氦嘴泄漏）
LD TR0
LD D1096.10  ; #2腔体机构开腔体氦检阀/延时关腔体抽气阀（自动步）
OR D1100.09  ; #2腔体机构开腔体氦检阀/延时关腔体抽气阀（自动单检步）
ANDLD
AND T2004  ; #2-1腔体氦检时间（测试）
OUT TR0
LD<=F(332) D302 D994  ; #2-1腔体测试漏率（Pa.m3/s_Float）, 泄漏率设定值（Pa.m3/s_Float）
OR H5.02  ; 氦检仪屏蔽
OR H5.10  ; 空跑程序
ANDLD
ANDNOT H31.00  ; #2-1电池泄漏
ANDNOT H31.02  ; #2-1电池注氦超时
ANDNOT H31.04  ; #2-1腔体抽真空NG
ANDNOT H31.06  ; #2-1腔体氦检时腔体压力过高
MOV(021) &1 D308  ; #2-1腔体测试结果（1 OK，2腔体泄漏，3气密NG，4注氦超时，5氦检异常，6电池泄漏，7注氦NG，8氦嘴泄漏）
LD TR0
AND>F(333) D302 D994  ; #2-1腔体测试漏率（Pa.m3/s_Float）, 泄漏率设定值（Pa.m3/s_Float）
ANDNOT H5.02  ; 氦检仪屏蔽
ANDNOT H5.10  ; 空跑程序
MOV(021) &3 D308  ; #2-1腔体测试结果（1 OK，2腔体泄漏，3气密NG，4注氦超时，5氦检异常，6电池泄漏，7注氦NG，8氦嘴泄漏）

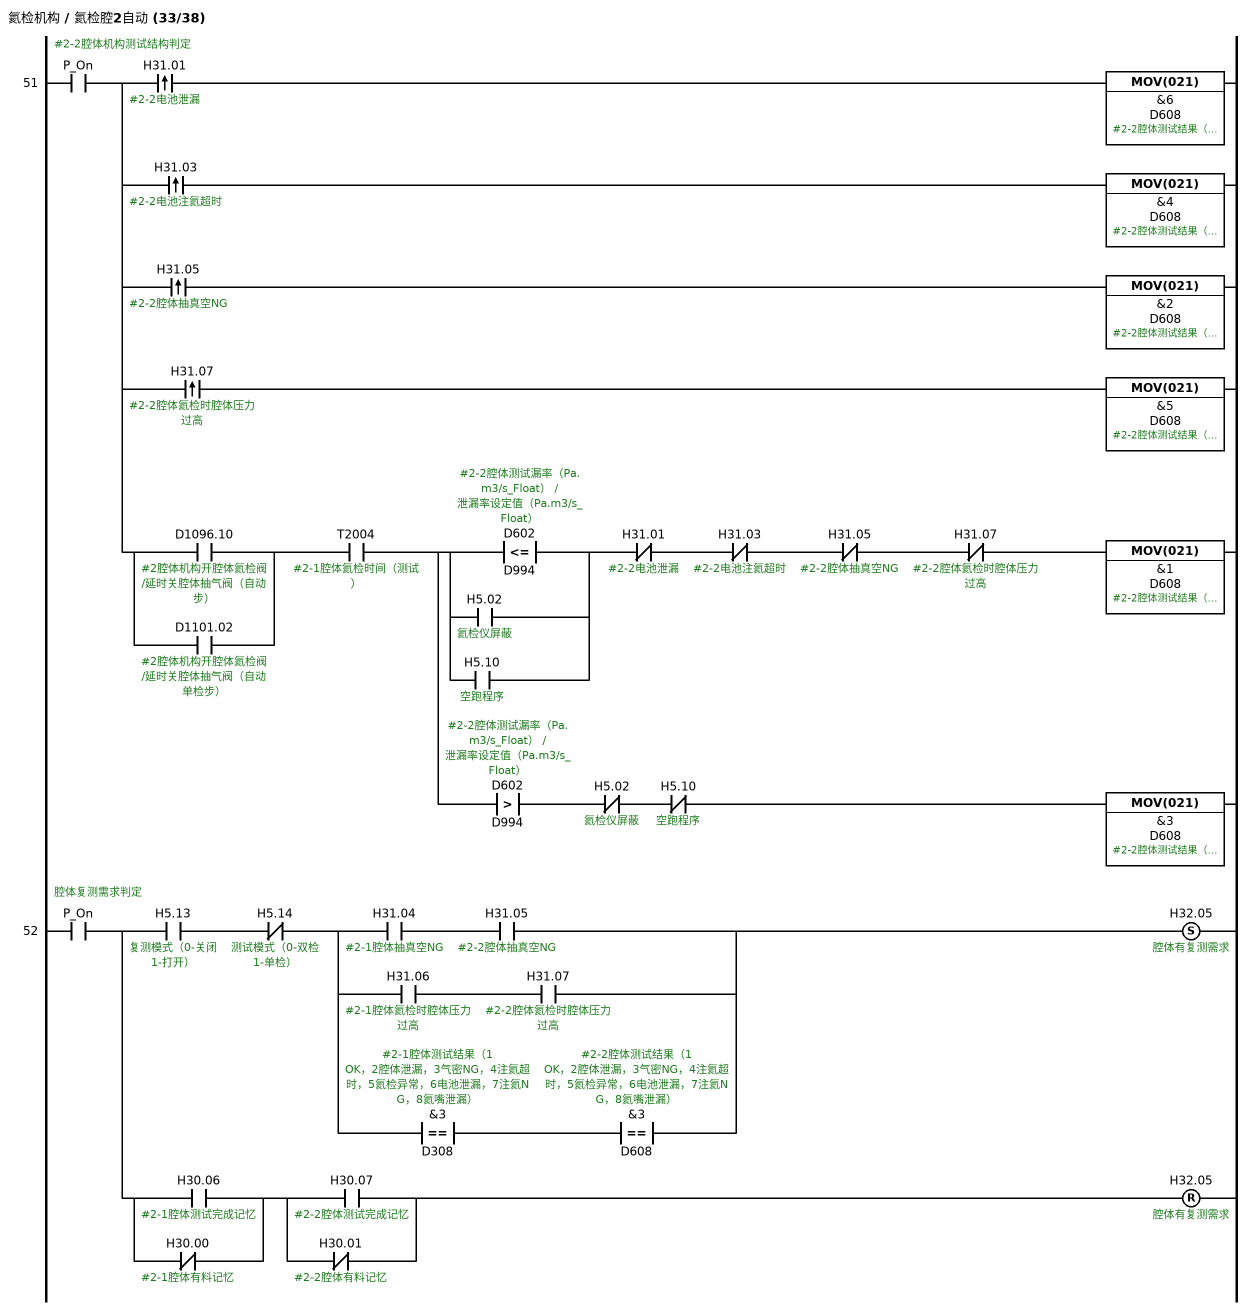
; rung 51: #2-2腔体机构测试结构判定
LD P_On
OUT TR0
@AND H31.01  ; #2-2电池泄漏
MOV(021) &6 D608  ; #2-2腔体测试结果（1 OK，2腔体泄漏，3气密NG，4注氦超时，5氦检异常，6电池泄漏，7注氦NG，8氦嘴泄漏）
LD TR0
@AND H31.03  ; #2-2电池注氦超时
MOV(021) &4 D608  ; #2-2腔体测试结果（1 OK，2腔体泄漏，3气密NG，4注氦超时，5氦检异常，6电池泄漏，7注氦NG，8氦嘴泄漏）
LD TR0
@AND H31.05  ; #2-2腔体抽真空NG
MOV(021) &2 D608  ; #2-2腔体测试结果（1 OK，2腔体泄漏，3气密NG，4注氦超时，5氦检异常，6电池泄漏，7注氦NG，8氦嘴泄漏）
LD TR0
@AND H31.07  ; #2-2腔体氦检时腔体压力过高
MOV(021) &5 D608  ; #2-2腔体测试结果（1 OK，2腔体泄漏，3气密NG，4注氦超时，5氦检异常，6电池泄漏，7注氦NG，8氦嘴泄漏）
LD TR0
LD D1096.10  ; #2腔体机构开腔体氦检阀/延时关腔体抽气阀（自动步）
OR D1101.02  ; #2腔体机构开腔体氦检阀/延时关腔体抽气阀（自动单检步）
ANDLD
AND T2004  ; #2-1腔体氦检时间（测试）
OUT TR0
LD<=F(332) D602 D994  ; #2-2腔体测试漏率（Pa.m3/s_Float）, 泄漏率设定值（Pa.m3/s_Float）
OR H5.02  ; 氦检仪屏蔽
OR H5.10  ; 空跑程序
ANDLD
ANDNOT H31.01  ; #2-2电池泄漏
ANDNOT H31.03  ; #2-2电池注氦超时
ANDNOT H31.05  ; #2-2腔体抽真空NG
ANDNOT H31.07  ; #2-2腔体氦检时腔体压力过高
MOV(021) &1 D608  ; #2-2腔体测试结果（1 OK，2腔体泄漏，3气密NG，4注氦超时，5氦检异常，6电池泄漏，7注氦NG，8氦嘴泄漏）
LD TR0
AND>F(333) D602 D994  ; #2-2腔体测试漏率（Pa.m3/s_Float）, 泄漏率设定值（Pa.m3/s_Float）
ANDNOT H5.02  ; 氦检仪屏蔽
ANDNOT H5.10  ; 空跑程序
MOV(021) &3 D608  ; #2-2腔体测试结果（1 OK，2腔体泄漏，3气密NG，4注氦超时，5氦检异常，6电池泄漏，7注氦NG，8氦嘴泄漏）
; rung 52: 腔体复测需求判定
LD P_On
OUT TR0
AND H5.13  ; 复测模式（0-关闭 1-打开）
ANDNOT H5.14  ; 测试模式（0-双检 1-单检）
LD H31.04  ; #2-1腔体抽真空NG
AND H31.05  ; #2-2腔体抽真空NG
LD H31.06  ; #2-1腔体氦检时腔体压力过高
AND H31.07  ; #2-2腔体氦检时腔体压力过高
ORLD
LD=(300) &3 D308  ; #2-1腔体测试结果（1 OK，2腔体泄漏，3气密NG，4注氦超时，5氦检异常，6电池泄漏，7注氦NG，8氦嘴泄漏）
AND=(300) &3 D608  ; #2-2腔体测试结果（1 OK，2腔体泄漏，3气密NG，4注氦超时，5氦检异常，6电池泄漏，7注氦NG，8氦嘴泄漏）
ORLD
ANDLD
SET H32.05  ; 腔体有复测需求
LD TR0
LD H30.06  ; #2-1腔体测试完成记忆
ORNOT H30.00  ; #2-1腔体有料记忆
ANDLD
LD H30.07  ; #2-2腔体测试完成记忆
ORNOT H30.01  ; #2-2腔体有料记忆
ANDLD
RSET H32.05  ; 腔体有复测需求

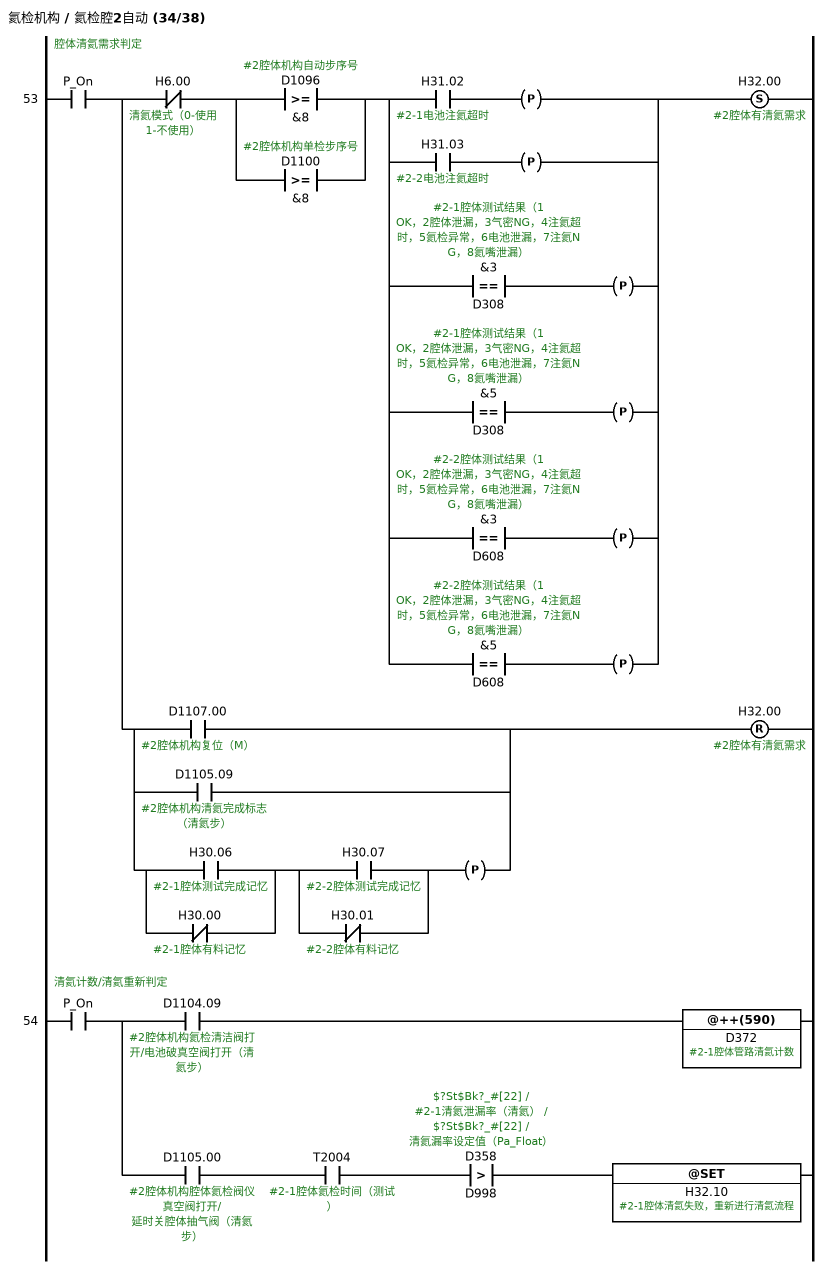
; rung 53: 腔体清氦需求判定
LD P_On
OUT TR0
ANDNOT H6.00  ; 清氦模式（0-使用 1-不使用）
LD>=L(326) D1096 &8  ; #2腔体机构自动步序号
OR>=L(326) D1100 &8  ; #2腔体机构单检步序号
ANDLD
LD H31.02  ; #2-1电池注氦超时
UP(521)
LD H31.03  ; #2-2电池注氦超时
UP(521)
ORLD
LD=(300) &3 D308  ; #2-1腔体测试结果（1 OK，2腔体泄漏，3气密NG，4注氦超时，5氦检异常，6电池泄漏，7注氦NG，8氦嘴泄漏）
UP(521)
ORLD
LD=(300) &5 D308  ; #2-1腔体测试结果（1 OK，2腔体泄漏，3气密NG，4注氦超时，5氦检异常，6电池泄漏，7注氦NG，8氦嘴泄漏）
UP(521)
ORLD
LD=(300) &3 D608  ; #2-2腔体测试结果（1 OK，2腔体泄漏，3气密NG，4注氦超时，5氦检异常，6电池泄漏，7注氦NG，8氦嘴泄漏）
UP(521)
ORLD
LD=(300) &5 D608  ; #2-2腔体测试结果（1 OK，2腔体泄漏，3气密NG，4注氦超时，5氦检异常，6电池泄漏，7注氦NG，8氦嘴泄漏）
UP(521)
ORLD
ANDLD
SET H32.00  ; #2腔体有清氦需求
LD TR0
LD D1107.00  ; #2腔体机构复位（M）
OR D1105.09  ; #2腔体机构清氦完成标志（清氦步）
LD H30.06  ; #2-1腔体测试完成记忆
ORNOT H30.00  ; #2-1腔体有料记忆
LD H30.07  ; #2-2腔体测试完成记忆
ORNOT H30.01  ; #2-2腔体有料记忆
ANDLD
UP(521)
ORLD
ANDLD
RSET H32.00  ; #2腔体有清氦需求
; rung 54: 清氦计数/清氦重新判定
LD P_On
OUT TR0
AND D1104.09  ; #2腔体机构氦检清洁阀打开/电池破真空阀打开（清氦步）
@++(590) D372  ; #2-1腔体管路清氦计数
LD TR0
AND D1105.00  ; #2腔体机构腔体氦检阀仪真空阀打开/延时关腔体抽气阀（清氦步）
AND T2004  ; #2-1腔体氦检时间（测试）
AND>F(333) D358 D998  ; $?St$Bk?_#[22] / #2-1清氦泄漏率（清氦） / $?St$Bk?_#[22], 清氦漏率设定值（Pa_Float）
@SET H32.10  ; #2-1腔体清氦失败，重新进行清氦流程

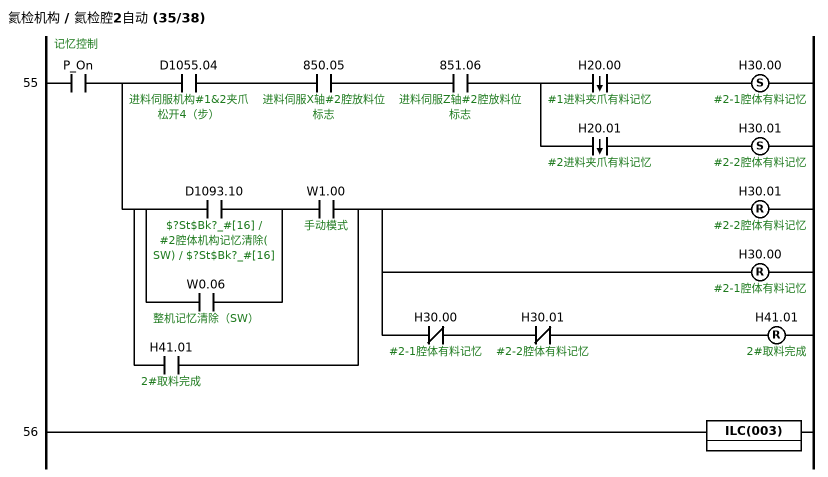
; rung 55: 记忆控制
LD P_On
OUT TR0
AND D1055.04  ; 进料伺服机构#1&2夹爪松开4（步）
AND 850.05  ; 进料伺服X轴#2腔放料位标志
AND 851.06  ; 进料伺服Z轴#2腔放料位标志
OUT TR1
%AND H20.00  ; #1进料夹爪有料记忆
SET H30.00  ; #2-1腔体有料记忆
LD TR1
%AND H20.01  ; #2进料夹爪有料记忆
SET H30.01  ; #2-2腔体有料记忆
LD TR0
LD D1093.10  ; $?St$Bk?_#[16] / #2腔体机构记忆清除(SW) / $?St$Bk?_#[16]
OR W0.06  ; 整机记忆清除（SW）
AND W1.00  ; 手动模式
OR H41.01  ; 2#取料完成
ANDLD
RSET H30.01  ; #2-2腔体有料记忆
RSET H30.00  ; #2-1腔体有料记忆
ANDNOT H30.00  ; #2-1腔体有料记忆
ANDNOT H30.01  ; #2-2腔体有料记忆
RSET H41.01  ; 2#取料完成
; rung 56
ILC(003)

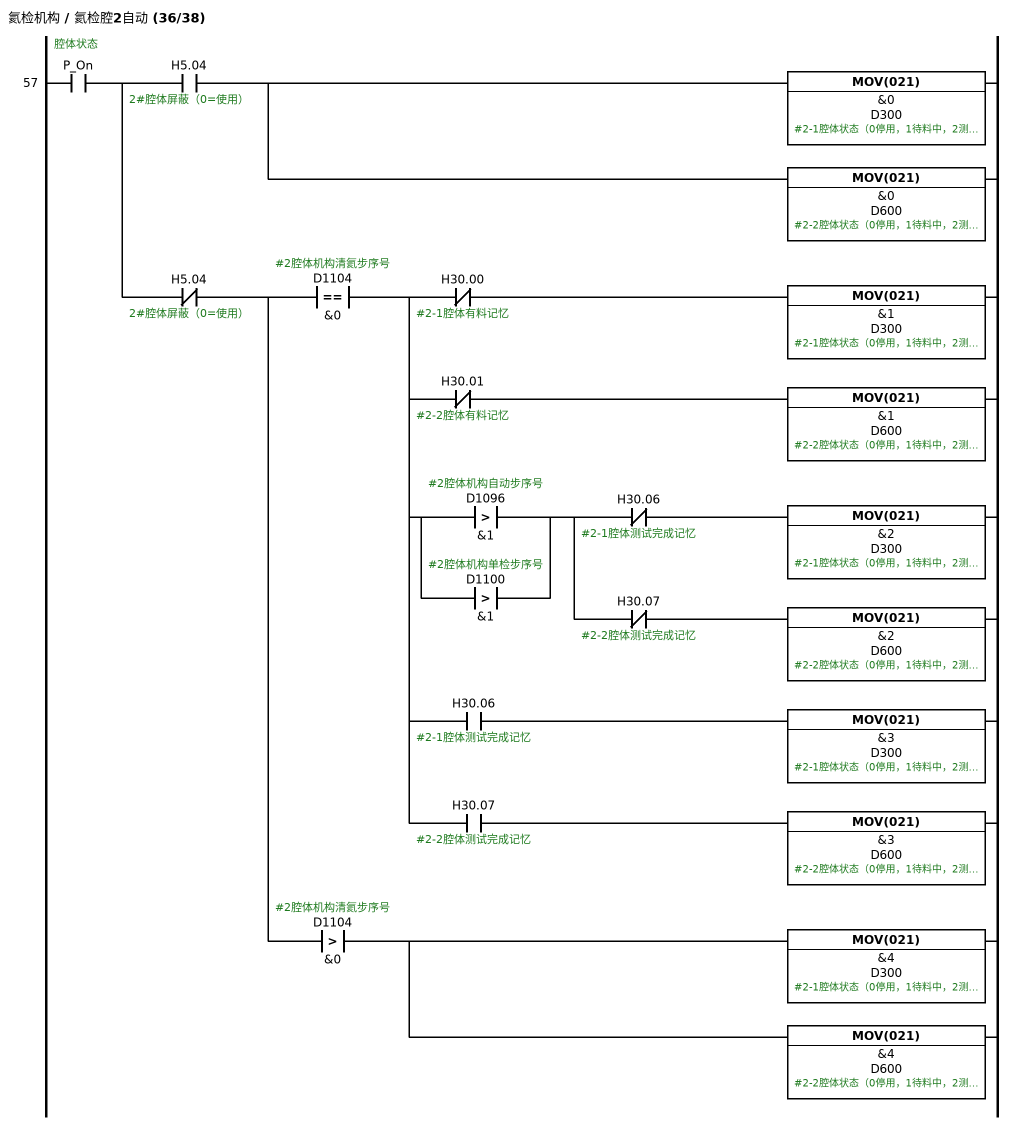
; rung 57: 腔体状态
LD P_On
OUT TR0
AND H5.04  ; 2#腔体屏蔽（0=使用）
MOV(021) &0 D300  ; #2-1腔体状态（0停用，1待料中，2测试中，3测试完成，4-清氦中）
MOV(021) &0 D600  ; #2-2腔体状态（0停用，1待料中，2测试中，3测试完成，4-清氦中）
LD TR0
ANDNOT H5.04  ; 2#腔体屏蔽（0=使用）
OUT TR0
AND=L(301) D1104 &0  ; #2腔体机构清氦步序号
OUT TR1
ANDNOT H30.00  ; #2-1腔体有料记忆
MOV(021) &1 D300  ; #2-1腔体状态（0停用，1待料中，2测试中，3测试完成，4-清氦中）
LD TR1
ANDNOT H30.01  ; #2-2腔体有料记忆
MOV(021) &1 D600  ; #2-2腔体状态（0停用，1待料中，2测试中，3测试完成，4-清氦中）
LD TR1
LD>L(321) D1096 &1  ; #2腔体机构自动步序号
OR>L(321) D1100 &1  ; #2腔体机构单检步序号
ANDLD
OUT TR2
ANDNOT H30.06  ; #2-1腔体测试完成记忆
MOV(021) &2 D300  ; #2-1腔体状态（0停用，1待料中，2测试中，3测试完成，4-清氦中）
LD TR2
ANDNOT H30.07  ; #2-2腔体测试完成记忆
MOV(021) &2 D600  ; #2-2腔体状态（0停用，1待料中，2测试中，3测试完成，4-清氦中）
LD TR1
AND H30.06  ; #2-1腔体测试完成记忆
MOV(021) &3 D300  ; #2-1腔体状态（0停用，1待料中，2测试中，3测试完成，4-清氦中）
LD TR1
AND H30.07  ; #2-2腔体测试完成记忆
MOV(021) &3 D600  ; #2-2腔体状态（0停用，1待料中，2测试中，3测试完成，4-清氦中）
LD TR0
AND>L(321) D1104 &0  ; #2腔体机构清氦步序号
MOV(021) &4 D300  ; #2-1腔体状态（0停用，1待料中，2测试中，3测试完成，4-清氦中）
MOV(021) &4 D600  ; #2-2腔体状态（0停用，1待料中，2测试中，3测试完成，4-清氦中）

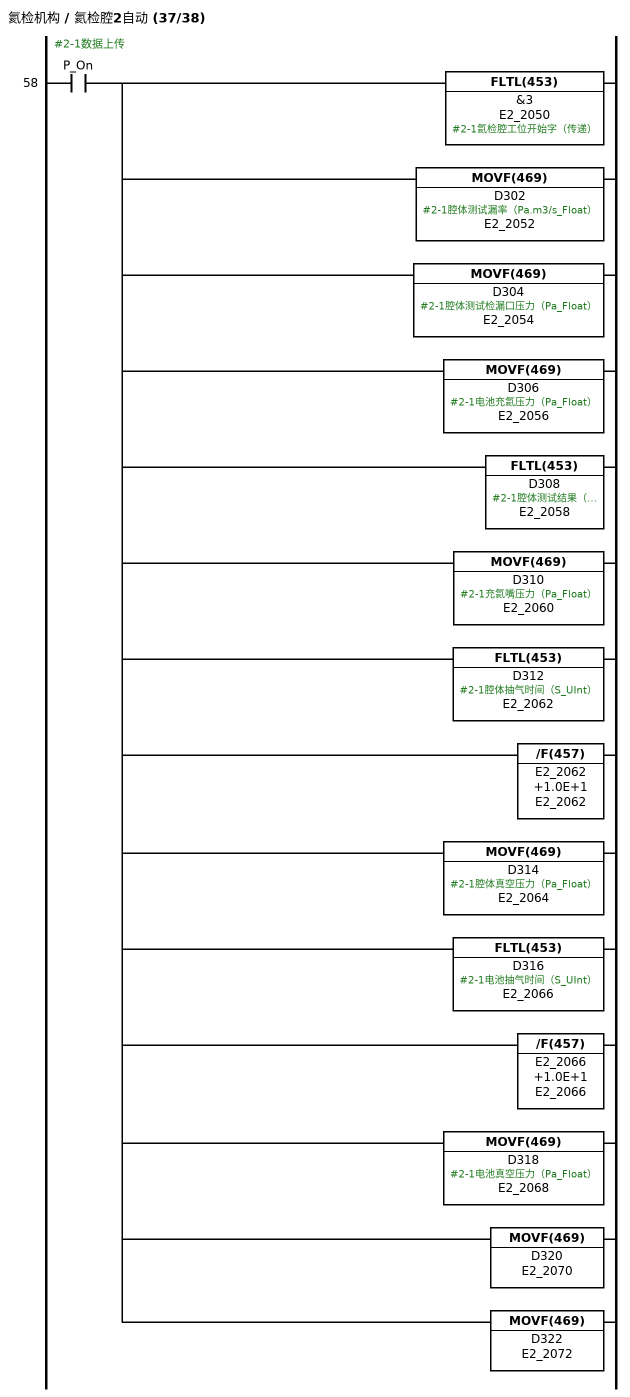
; rung 58: #2-1数据上传
LD P_On
FLTL(453) &3 E2_2050  ; #2-1氦检腔工位开始字（传递）
MOVF(469) D302 E2_2052  ; #2-1腔体测试漏率（Pa.m3/s_Float）
MOVF(469) D304 E2_2054  ; #2-1腔体测试检漏口压力（Pa_Float）
MOVF(469) D306 E2_2056  ; #2-1电池充氦压力（Pa_Float）
FLTL(453) D308 E2_2058  ; #2-1腔体测试结果（1 OK，2腔体泄漏，3气密NG，4注氦超时，5氦检异常，6电池泄漏，7注氦NG，8氦嘴泄漏）
MOVF(469) D310 E2_2060  ; #2-1充氦嘴压力（Pa_Float）
FLTL(453) D312 E2_2062  ; #2-1腔体抽气时间（S_UInt）
/F(457) E2_2062 +1.0E+1 E2_2062
MOVF(469) D314 E2_2064  ; #2-1腔体真空压力（Pa_Float）
FLTL(453) D316 E2_2066  ; #2-1电池抽气时间（S_UInt）
/F(457) E2_2066 +1.0E+1 E2_2066
MOVF(469) D318 E2_2068  ; #2-1电池真空压力（Pa_Float）
MOVF(469) D320 E2_2070
MOVF(469) D322 E2_2072

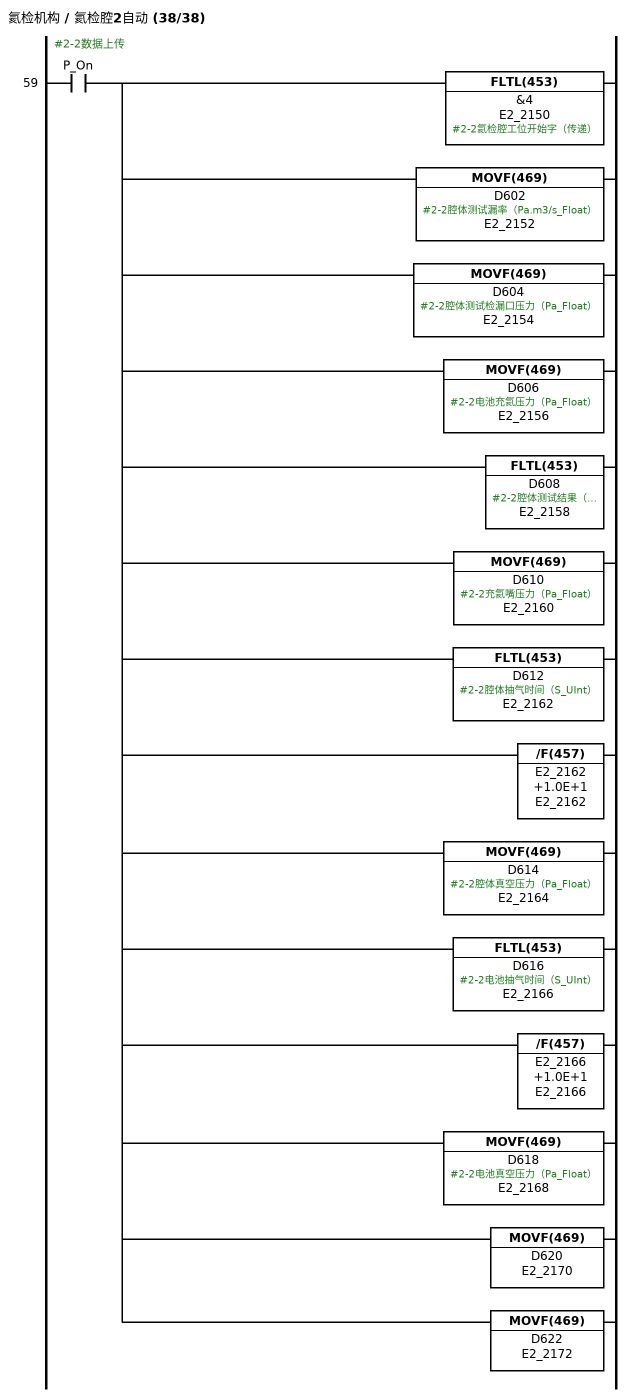
; rung 59: #2-2数据上传
LD P_On
FLTL(453) &4 E2_2150  ; #2-2氦检腔工位开始字（传递）
MOVF(469) D602 E2_2152  ; #2-2腔体测试漏率（Pa.m3/s_Float）
MOVF(469) D604 E2_2154  ; #2-2腔体测试检漏口压力（Pa_Float）
MOVF(469) D606 E2_2156  ; #2-2电池充氦压力（Pa_Float）
FLTL(453) D608 E2_2158  ; #2-2腔体测试结果（1 OK，2腔体泄漏，3气密NG，4注氦超时，5氦检异常，6电池泄漏，7注氦NG，8氦嘴泄漏）
MOVF(469) D610 E2_2160  ; #2-2充氦嘴压力（Pa_Float）
FLTL(453) D612 E2_2162  ; #2-2腔体抽气时间（S_UInt）
/F(457) E2_2162 +1.0E+1 E2_2162
MOVF(469) D614 E2_2164  ; #2-2腔体真空压力（Pa_Float）
FLTL(453) D616 E2_2166  ; #2-2电池抽气时间（S_UInt）
/F(457) E2_2166 +1.0E+1 E2_2166
MOVF(469) D618 E2_2168  ; #2-2电池真空压力（Pa_Float）
MOVF(469) D620 E2_2170
MOVF(469) D622 E2_2172

### Section 氦检腔3自动

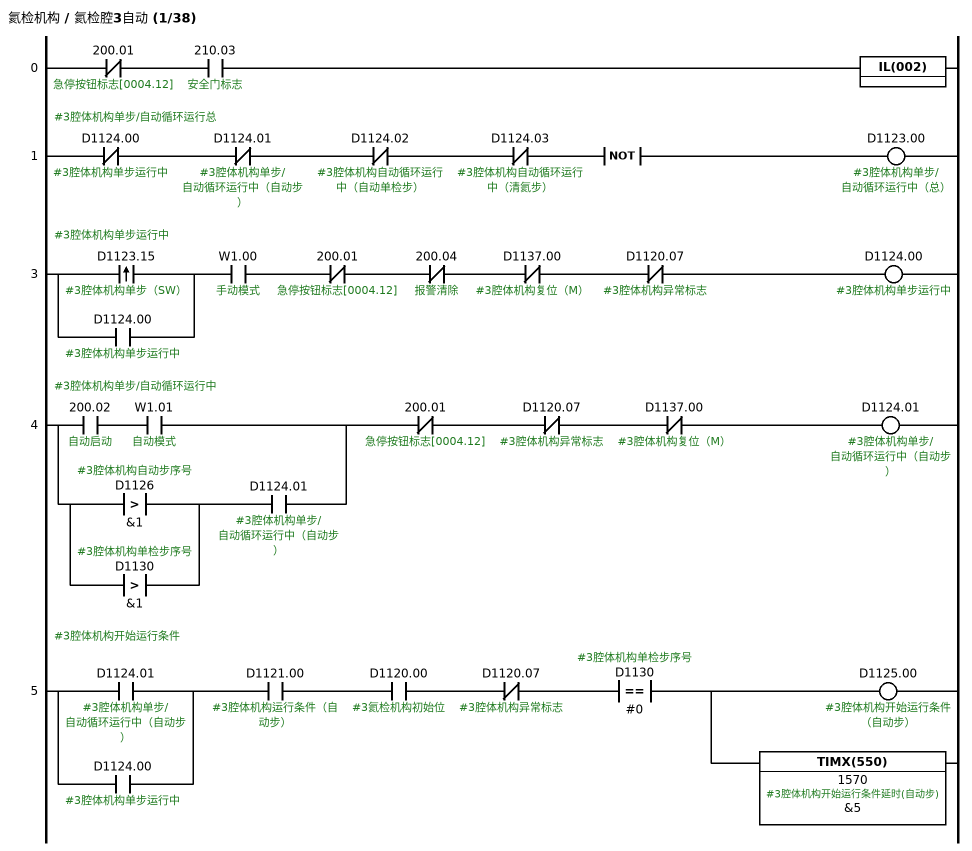
; rung 0
LDNOT 200.01  ; 急停按钮标志[0004.12]
AND 210.03  ; 安全门标志
IL(002)
; rung 1: #3腔体机构单步/自动循环运行总
LDNOT D1124.00  ; #3腔体机构单步运行中
ANDNOT D1124.01  ; #3腔体机构单步/自动循环运行中（自动步）
ANDNOT D1124.02  ; #3腔体机构自动循环运行中（自动单检步）
ANDNOT D1124.03  ; #3腔体机构自动循环运行中（清氦步）
NOT(520)
OUT D1123.00  ; #3腔体机构单步/自动循环运行中（总）
; rung 2: ******************************* / 自动双检步序 / *******************************
; rung 3: #3腔体机构单步运行中
@LD D1123.15  ; #3腔体机构单步（SW）
OR D1124.00  ; #3腔体机构单步运行中
AND W1.00  ; 手动模式
ANDNOT 200.01  ; 急停按钮标志[0004.12]
ANDNOT 200.04  ; 报警清除
ANDNOT D1137.00  ; #3腔体机构复位（M）
ANDNOT D1120.07  ; #3腔体机构异常标志
OUT D1124.00  ; #3腔体机构单步运行中
; rung 4: #3腔体机构单步/自动循环运行中
LD 200.02  ; 自动启动
AND W1.01  ; 自动模式
LD>L(321) D1126 &1  ; #3腔体机构自动步序号
OR>L(321) D1130 &1  ; #3腔体机构单检步序号
AND D1124.01  ; #3腔体机构单步/自动循环运行中（自动步）
ORLD
ANDNOT 200.01  ; 急停按钮标志[0004.12]
ANDNOT D1120.07  ; #3腔体机构异常标志
ANDNOT D1137.00  ; #3腔体机构复位（M）
OUT D1124.01  ; #3腔体机构单步/自动循环运行中（自动步）
; rung 5: #3腔体机构开始运行条件
LD D1124.01  ; #3腔体机构单步/自动循环运行中（自动步）
OR D1124.00  ; #3腔体机构单步运行中
AND D1121.00  ; #3腔体机构运行条件（自动步）
AND D1120.00  ; #3氦检机构初始位
ANDNOT D1120.07  ; #3腔体机构异常标志
AND=L(301) D1130 #0  ; #3腔体机构单检步序号
OUT D1125.00  ; #3腔体机构开始运行条件（自动步）
TIMX(550) 1570 &5  ; #3腔体机构开始运行条件延时(自动步)

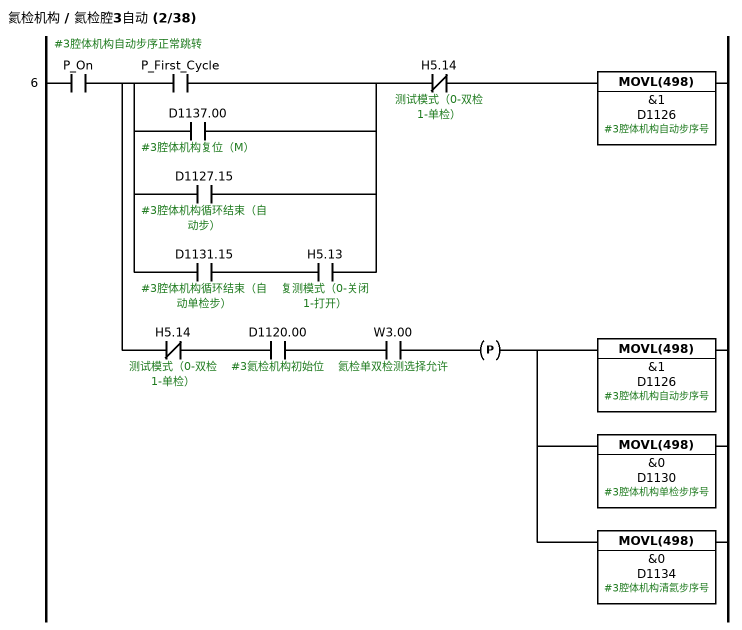
; rung 6: #3腔体机构自动步序正常跳转
LD P_On
OUT TR0
LD P_First_Cycle
OR D1137.00  ; #3腔体机构复位（M）
OR D1127.15  ; #3腔体机构循环结束（自动步）
LD D1131.15  ; #3腔体机构循环结束（自动单检步）
AND H5.13  ; 复测模式（0-关闭 1-打开）
ORLD
ANDLD
ANDNOT H5.14  ; 测试模式（0-双检 1-单检）
MOVL(498) &1 D1126  ; #3腔体机构自动步序号
LD TR0
ANDNOT H5.14  ; 测试模式（0-双检 1-单检）
AND D1120.00  ; #3氦检机构初始位
AND W3.00  ; 氦检单双检测选择允许
UP(521)
MOVL(498) &1 D1126  ; #3腔体机构自动步序号
MOVL(498) &0 D1130  ; #3腔体机构单检步序号
MOVL(498) &0 D1134  ; #3腔体机构清氦步序号

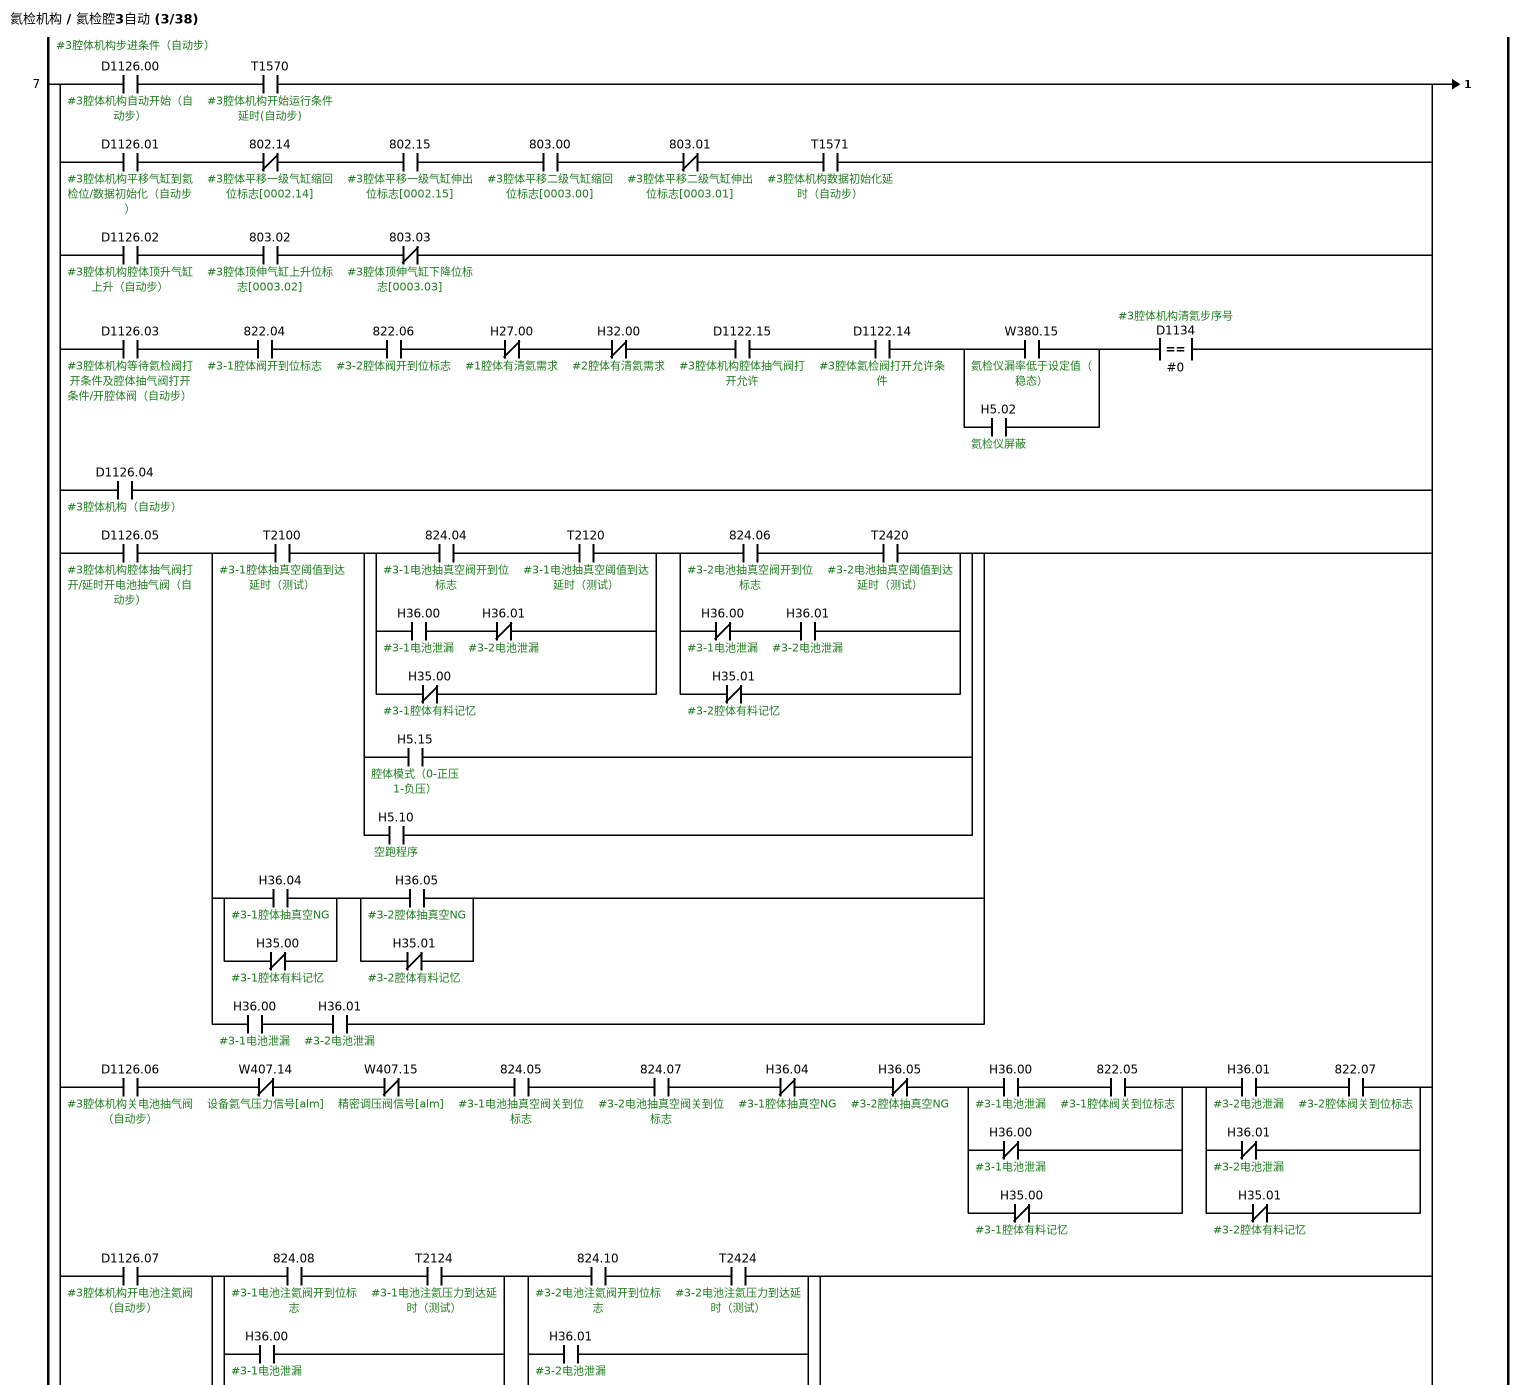

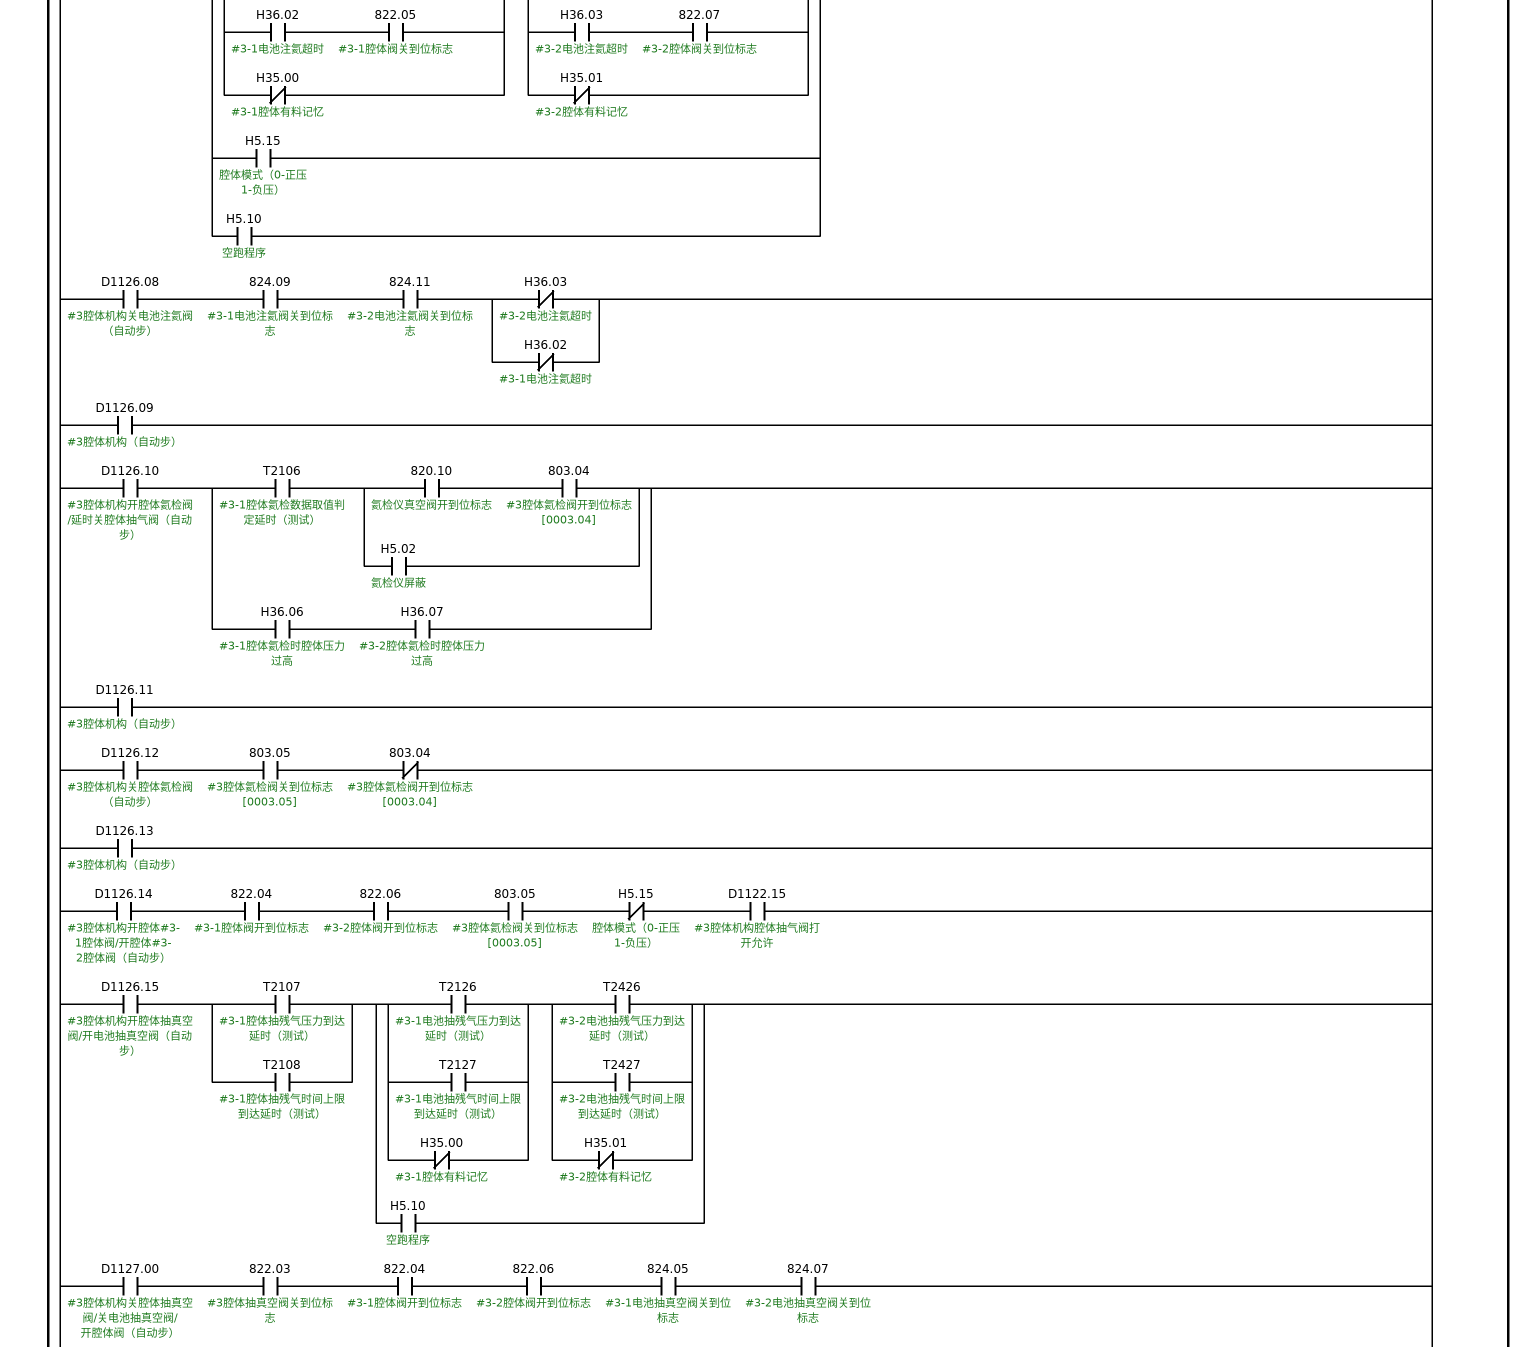

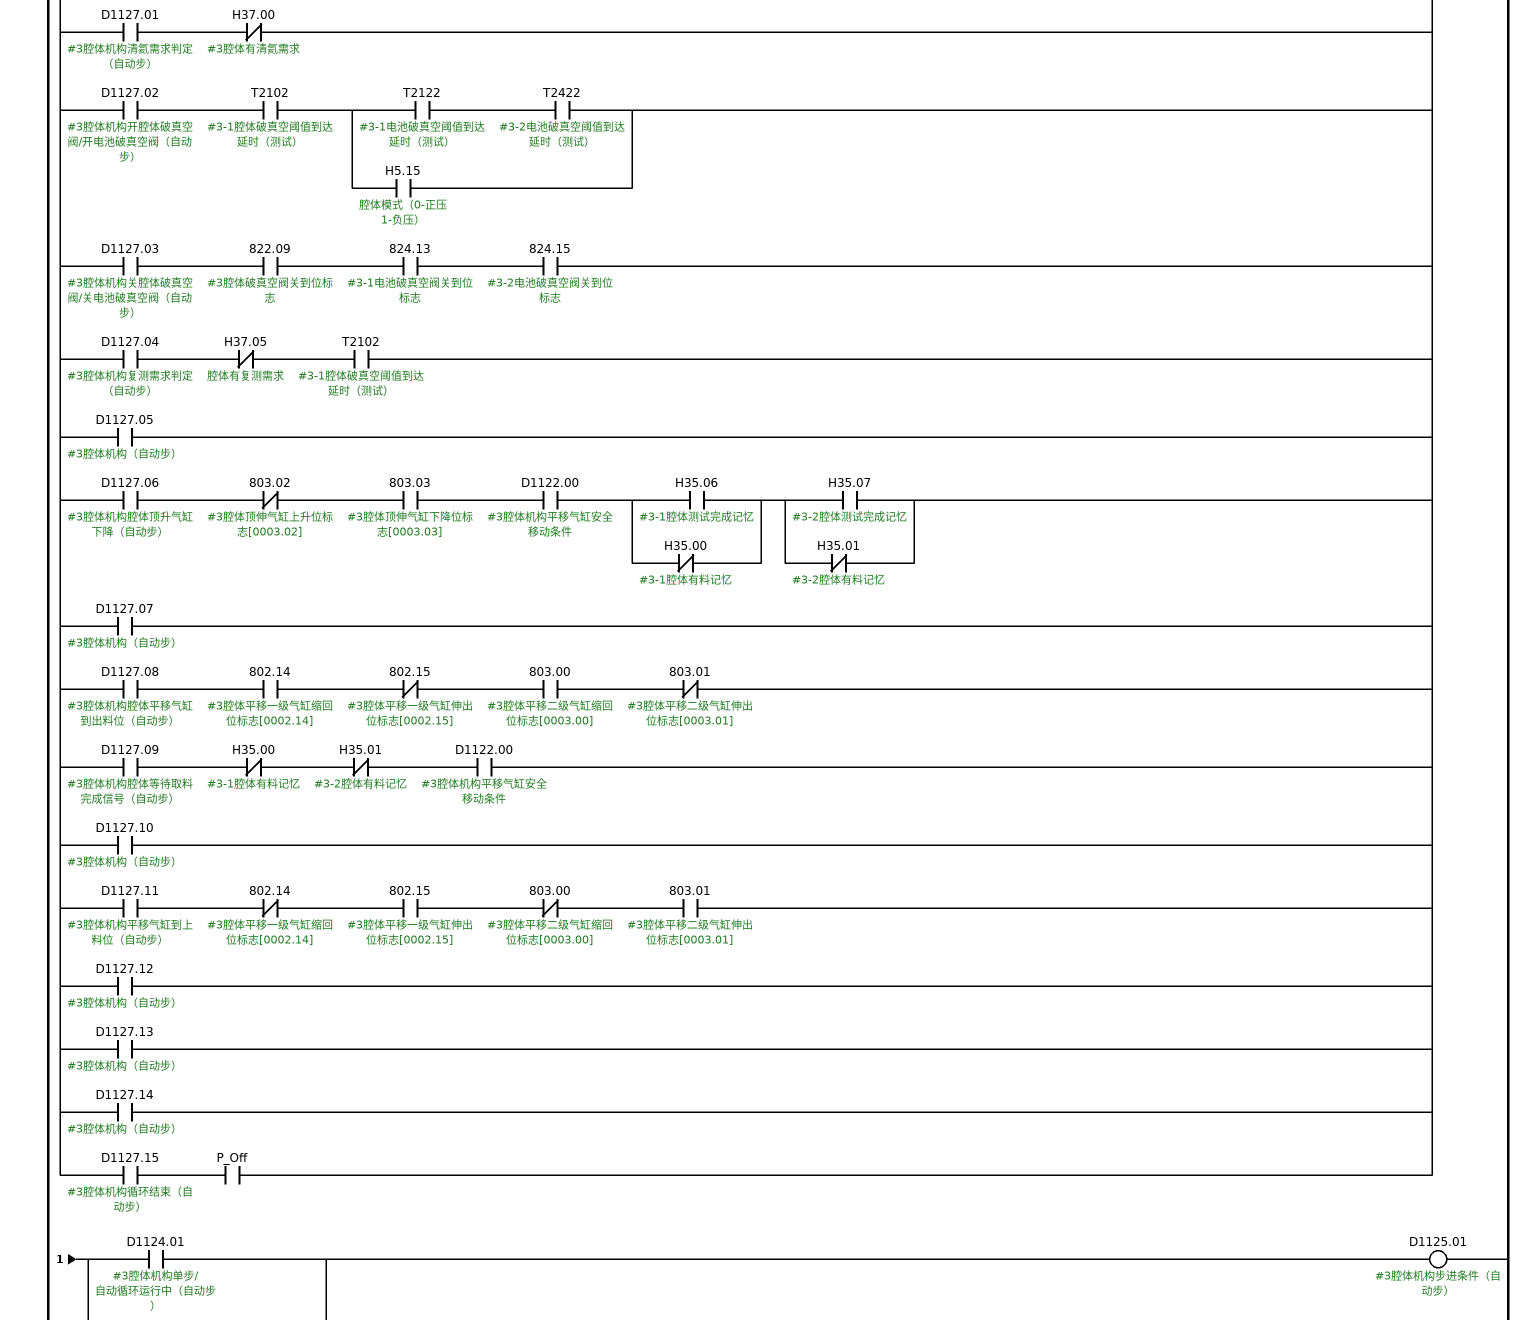

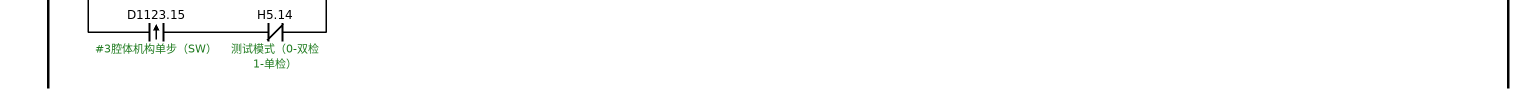
; rung 7: #3腔体机构步进条件（自动步）
LD D1126.00  ; #3腔体机构自动开始（自动步）
AND T1570  ; #3腔体机构开始运行条件延时(自动步)
LD D1126.01  ; #3腔体机构平移气缸到氦检位/数据初始化（自动步）
ANDNOT 802.14  ; #3腔体平移一级气缸缩回位标志[0002.14]
AND 802.15  ; #3腔体平移一级气缸伸出位标志[0002.15]
AND 803.00  ; #3腔体平移二级气缸缩回位标志[0003.00]
ANDNOT 803.01  ; #3腔体平移二级气缸伸出位标志[0003.01]
AND T1571  ; #3腔体机构数据初始化延时（自动步）
ORLD
LD D1126.02  ; #3腔体机构腔体顶升气缸上升（自动步）
AND 803.02  ; #3腔体顶伸气缸上升位标志[0003.02]
ANDNOT 803.03  ; #3腔体顶伸气缸下降位标志[0003.03]
ORLD
LD D1126.03  ; #3腔体机构等待氦检阀打开条件及腔体抽气阀打开条件/开腔体阀（自动步）
AND 822.04  ; #3-1腔体阀开到位标志
AND 822.06  ; #3-2腔体阀开到位标志
ANDNOT H27.00  ; #1腔体有清氦需求
ANDNOT H32.00  ; #2腔体有清氦需求
AND D1122.15  ; #3腔体机构腔体抽气阀打开允许
AND D1122.14  ; #3腔体氦检阀打开允许条件
LD W380.15  ; 氦检仪漏率低于设定值（稳态）
OR H5.02  ; 氦检仪屏蔽
ANDLD
AND=L(301) D1134 #0  ; #3腔体机构清氦步序号
ORLD
OR D1126.04  ; #3腔体机构（自动步）
LD D1126.05  ; #3腔体机构腔体抽气阀打开/延时开电池抽气阀（自动步）
LD T2100  ; #3-1腔体抽真空阈值到达延时（测试）
LD 824.04  ; #3-1电池抽真空阀开到位标志
AND T2120  ; #3-1电池抽真空阈值到达延时（测试）
LD H36.00  ; #3-1电池泄漏
ANDNOT H36.01  ; #3-2电池泄漏
ORLD
ORNOT H35.00  ; #3-1腔体有料记忆
LD 824.06  ; #3-2电池抽真空阀开到位标志
AND T2420  ; #3-2电池抽真空阈值到达延时（测试）
LDNOT H36.00  ; #3-1电池泄漏
AND H36.01  ; #3-2电池泄漏
ORLD
ORNOT H35.01  ; #3-2腔体有料记忆
ANDLD
OR H5.15  ; 腔体模式（0-正压 1-负压）
OR H5.10  ; 空跑程序
ANDLD
LD H36.04  ; #3-1腔体抽真空NG
ORNOT H35.00  ; #3-1腔体有料记忆
LD H36.05  ; #3-2腔体抽真空NG
ORNOT H35.01  ; #3-2腔体有料记忆
ANDLD
ORLD
LD H36.00  ; #3-1电池泄漏
AND H36.01  ; #3-2电池泄漏
ORLD
ANDLD
ORLD
LD D1126.06  ; #3腔体机构关电池抽气阀（自动步）  // 单个电池出现电池泄漏时，需将对应的腔体阀门关闭
ANDNOT W407.14  ; 设备氦气压力信号[alm]
ANDNOT W407.15  ; 精密调压阀信号[alm]
AND 824.05  ; #3-1电池抽真空阀关到位标志
AND 824.07  ; #3-2电池抽真空阀关到位标志
ANDNOT H36.04  ; #3-1腔体抽真空NG
ANDNOT H36.05  ; #3-2腔体抽真空NG
LD H36.00  ; #3-1电池泄漏
AND 822.05  ; #3-1腔体阀关到位标志
ORNOT H36.00  ; #3-1电池泄漏
ORNOT H35.00  ; #3-1腔体有料记忆
ANDLD
LD H36.01  ; #3-2电池泄漏
AND 822.07  ; #3-2腔体阀关到位标志
ORNOT H36.01  ; #3-2电池泄漏
ORNOT H35.01  ; #3-2腔体有料记忆
ANDLD
ORLD
LD D1126.07  ; #3腔体机构开电池注氦阀（自动步）  // 单个电池出现注氦超时时，需将对应的腔体阀门关闭
LD 824.08  ; #3-1电池注氦阀开到位标志
AND T2124  ; #3-1电池注氦压力到达延时（测试）
OR H36.00  ; #3-1电池泄漏
LD H36.02  ; #3-1电池注氦超时
AND 822.05  ; #3-1腔体阀关到位标志
ORLD
ORNOT H35.00  ; #3-1腔体有料记忆
LD 824.10  ; #3-2电池注氦阀开到位标志
AND T2424  ; #3-2电池注氦压力到达延时（测试）
OR H36.01  ; #3-2电池泄漏
LD H36.03  ; #3-2电池注氦超时
AND 822.07  ; #3-2腔体阀关到位标志
ORLD
ORNOT H35.01  ; #3-2腔体有料记忆
ANDLD
OR H5.15  ; 腔体模式（0-正压 1-负压）
OR H5.10  ; 空跑程序
ANDLD
ORLD
LD D1126.08  ; #3腔体机构关电池注氦阀（自动步）
AND 824.09  ; #3-1电池注氦阀关到位标志
AND 824.11  ; #3-2电池注氦阀关到位标志
LDNOT H36.03  ; #3-2电池注氦超时
ORNOT H36.02  ; #3-1电池注氦超时
ANDLD
ORLD
OR D1126.09  ; #3腔体机构（自动步）
LD D1126.10  ; #3腔体机构开腔体氦检阀/延时关腔体抽气阀（自动步）
LD T2106  ; #3-1腔体氦检数据取值判定延时（测试）
LD 820.10  ; 氦检仪真空阀开到位标志
AND 803.04  ; #3腔体氦检阀开到位标志[0003.04]
OR H5.02  ; 氦检仪屏蔽
ANDLD
LD H36.06  ; #3-1腔体氦检时腔体压力过高
AND H36.07  ; #3-2腔体氦检时腔体压力过高
ORLD
ANDLD
ORLD
OR D1126.11  ; #3腔体机构（自动步）
LD D1126.12  ; #3腔体机构关腔体氦检阀（自动步）
AND 803.05  ; #3腔体氦检阀关到位标志[0003.05]
ANDNOT 803.04  ; #3腔体氦检阀开到位标志[0003.04]
ORLD
OR D1126.13  ; #3腔体机构（自动步）
LD D1126.14  ; #3腔体机构开腔体#3-1腔体阀/开腔体#3-2腔体阀（自动步）
AND 822.04  ; #3-1腔体阀开到位标志
AND 822.06  ; #3-2腔体阀开到位标志
AND 803.05  ; #3腔体氦检阀关到位标志[0003.05]
ANDNOT H5.15  ; 腔体模式（0-正压 1-负压）
AND D1122.15  ; #3腔体机构腔体抽气阀打开允许
ORLD
LD D1126.15  ; #3腔体机构开腔体抽真空阀/开电池抽真空阀（自动步）
LD T2107  ; #3-1腔体抽残气压力到达延时（测试）
OR T2108  ; #3-1腔体抽残气时间上限到达延时（测试）
ANDLD
LD T2126  ; #3-1电池抽残气压力到达延时（测试）
OR T2127  ; #3-1电池抽残气时间上限到达延时（测试）
ORNOT H35.00  ; #3-1腔体有料记忆
LD T2426  ; #3-2电池抽残气压力到达延时（测试）
OR T2427  ; #3-2电池抽残气时间上限到达延时（测试）
ORNOT H35.01  ; #3-2腔体有料记忆
ANDLD
OR H5.10  ; 空跑程序
ANDLD
ORLD
LD D1127.00  ; #3腔体机构关腔体抽真空阀/关电池抽真空阀/开腔体阀（自动步）
AND 822.03  ; #3腔体抽真空阀关到位标志
AND 822.04  ; #3-1腔体阀开到位标志
AND 822.06  ; #3-2腔体阀开到位标志
AND 824.05  ; #3-1电池抽真空阀关到位标志
AND 824.07  ; #3-2电池抽真空阀关到位标志
ORLD
LD D1127.01  ; #3腔体机构清氦需求判定（自动步）
ANDNOT H37.00  ; #3腔体有清氦需求
ORLD
LD D1127.02  ; #3腔体机构开腔体破真空阀/开电池破真空阀（自动步）
AND T2102  ; #3-1腔体破真空阈值到达延时（测试）
LD T2122  ; #3-1电池破真空阈值到达延时（测试）
AND T2422  ; #3-2电池破真空阈值到达延时（测试）
OR H5.15  ; 腔体模式（0-正压 1-负压）
ANDLD
ORLD
LD D1127.03  ; #3腔体机构关腔体破真空阀/关电池破真空阀（自动步）
AND 822.09  ; #3腔体破真空阀关到位标志
AND 824.13  ; #3-1电池破真空阀关到位标志
AND 824.15  ; #3-2电池破真空阀关到位标志
ORLD
LD D1127.04  ; #3腔体机构复测需求判定（自动步）
ANDNOT H37.05  ; 腔体有复测需求
AND T2102  ; #3-1腔体破真空阈值到达延时（测试）
ORLD
OR D1127.05  ; #3腔体机构（自动步）
LD D1127.06  ; #3腔体机构腔体顶升气缸下降（自动步）
ANDNOT 803.02  ; #3腔体顶伸气缸上升位标志[0003.02]
AND 803.03  ; #3腔体顶伸气缸下降位标志[0003.03]
AND D1122.00  ; #3腔体机构平移气缸安全移动条件
LD H35.06  ; #3-1腔体测试完成记忆
ORNOT H35.00  ; #3-1腔体有料记忆
ANDLD
LD H35.07  ; #3-2腔体测试完成记忆
ORNOT H35.01  ; #3-2腔体有料记忆
ANDLD
ORLD
OR D1127.07  ; #3腔体机构（自动步）
LD D1127.08  ; #3腔体机构腔体平移气缸到出料位（自动步）
AND 802.14  ; #3腔体平移一级气缸缩回位标志[0002.14]
ANDNOT 802.15  ; #3腔体平移一级气缸伸出位标志[0002.15]
AND 803.00  ; #3腔体平移二级气缸缩回位标志[0003.00]
ANDNOT 803.01  ; #3腔体平移二级气缸伸出位标志[0003.01]
ORLD
LD D1127.09  ; #3腔体机构腔体等待取料完成信号（自动步）
ANDNOT H35.00  ; #3-1腔体有料记忆
ANDNOT H35.01  ; #3-2腔体有料记忆
AND D1122.00  ; #3腔体机构平移气缸安全移动条件
ORLD
OR D1127.10  ; #3腔体机构（自动步）
LD D1127.11  ; #3腔体机构平移气缸到上料位（自动步）
ANDNOT 802.14  ; #3腔体平移一级气缸缩回位标志[0002.14]
AND 802.15  ; #3腔体平移一级气缸伸出位标志[0002.15]
ANDNOT 803.00  ; #3腔体平移二级气缸缩回位标志[0003.00]
AND 803.01  ; #3腔体平移二级气缸伸出位标志[0003.01]
ORLD
OR D1127.12  ; #3腔体机构（自动步）
OR D1127.13  ; #3腔体机构（自动步）
OR D1127.14  ; #3腔体机构（自动步）
LD D1127.15  ; #3腔体机构循环结束（自动步）
AND P_Off
ORLD
LD D1124.01  ; #3腔体机构单步/自动循环运行中（自动步）
@LD D1123.15  ; #3腔体机构单步（SW）
ANDNOT H5.14  ; 测试模式（0-双检 1-单检）
ORLD
ANDLD
OUT D1125.01  ; #3腔体机构步进条件（自动步）

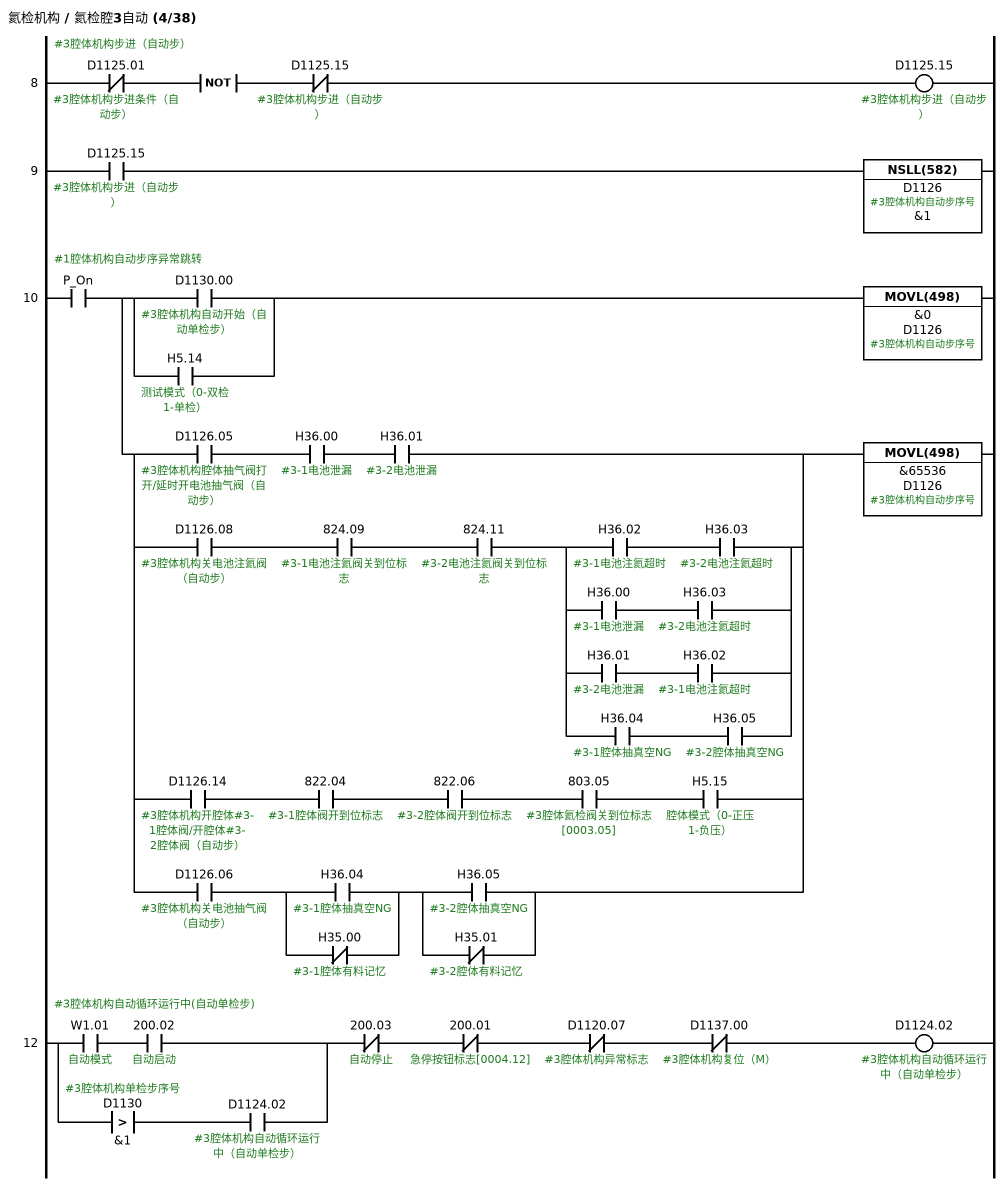
; rung 8: #3腔体机构步进（自动步）
LDNOT D1125.01  ; #3腔体机构步进条件（自动步）
NOT(520)
ANDNOT D1125.15  ; #3腔体机构步进（自动步）
OUT D1125.15  ; #3腔体机构步进（自动步）
; rung 9
LD D1125.15  ; #3腔体机构步进（自动步）
NSLL(582) D1126 &1  ; #3腔体机构自动步序号
; rung 10: #1腔体机构自动步序异常跳转
LD P_On
OUT TR0
LD D1130.00  ; #3腔体机构自动开始（自动单检步）
OR H5.14  ; 测试模式（0-双检 1-单检）
ANDLD
MOVL(498) &0 D1126  ; #3腔体机构自动步序号  // 测试模式为单检模式，腔体进入到复测步序时，将腔体机构自动步序清零
LD TR0
LD D1126.05  ; #3腔体机构腔体抽气阀打开/延时开电池抽气阀（自动步）
AND H36.00  ; #3-1电池泄漏
AND H36.01  ; #3-2电池泄漏
LD D1126.08  ; #3腔体机构关电池注氦阀（自动步）
AND 824.09  ; #3-1电池注氦阀关到位标志
AND 824.11  ; #3-2电池注氦阀关到位标志
LD H36.02  ; #3-1电池注氦超时
AND H36.03  ; #3-2电池注氦超时
LD H36.00  ; #3-1电池泄漏
AND H36.03  ; #3-2电池注氦超时
ORLD
LD H36.01  ; #3-2电池泄漏
AND H36.02  ; #3-1电池注氦超时
ORLD
LD H36.04  ; #3-1腔体抽真空NG
AND H36.05  ; #3-2腔体抽真空NG
ORLD
ANDLD
ORLD
LD D1126.14  ; #3腔体机构开腔体#3-1腔体阀/开腔体#3-2腔体阀（自动步）  // 负压模式不需要进行氦检后抽真空动作
AND 822.04  ; #3-1腔体阀开到位标志
AND 822.06  ; #3-2腔体阀开到位标志
AND 803.05  ; #3腔体氦检阀关到位标志[0003.05]
AND H5.15  ; 腔体模式（0-正压 1-负压）
ORLD
LD D1126.06  ; #3腔体机构关电池抽气阀（自动步）
LD H36.04  ; #3-1腔体抽真空NG
ORNOT H35.00  ; #3-1腔体有料记忆
ANDLD
LD H36.05  ; #3-2腔体抽真空NG
ORNOT H35.01  ; #3-2腔体有料记忆
ANDLD
ORLD
ANDLD
MOVL(498) &65536 D1126  ; #3腔体机构自动步序号  // 出现腔体抽真空NG，双电池抽真空NG，双电池注氦超时的情况，均跳转至自动步序D1067.0
; rung 11: ******************************* / 自动单检步序 / *******************************
; rung 12: #3腔体机构自动循环运行中(自动单检步)
LD W1.01  ; 自动模式
AND 200.02  ; 自动启动
LD>L(321) D1130 &1  ; #3腔体机构单检步序号
AND D1124.02  ; #3腔体机构自动循环运行中（自动单检步）
ORLD
ANDNOT 200.03  ; 自动停止
ANDNOT 200.01  ; 急停按钮标志[0004.12]
ANDNOT D1120.07  ; #3腔体机构异常标志
ANDNOT D1137.00  ; #3腔体机构复位（M）
OUT D1124.02  ; #3腔体机构自动循环运行中（自动单检步）

